// Mitsubishi GX Works2 project: GBOV-76_20100001_210617 H   PLC: Q06UDV
// 21/3/19(五)_進料手臂/開爪修正_

PROGRAM SERVO
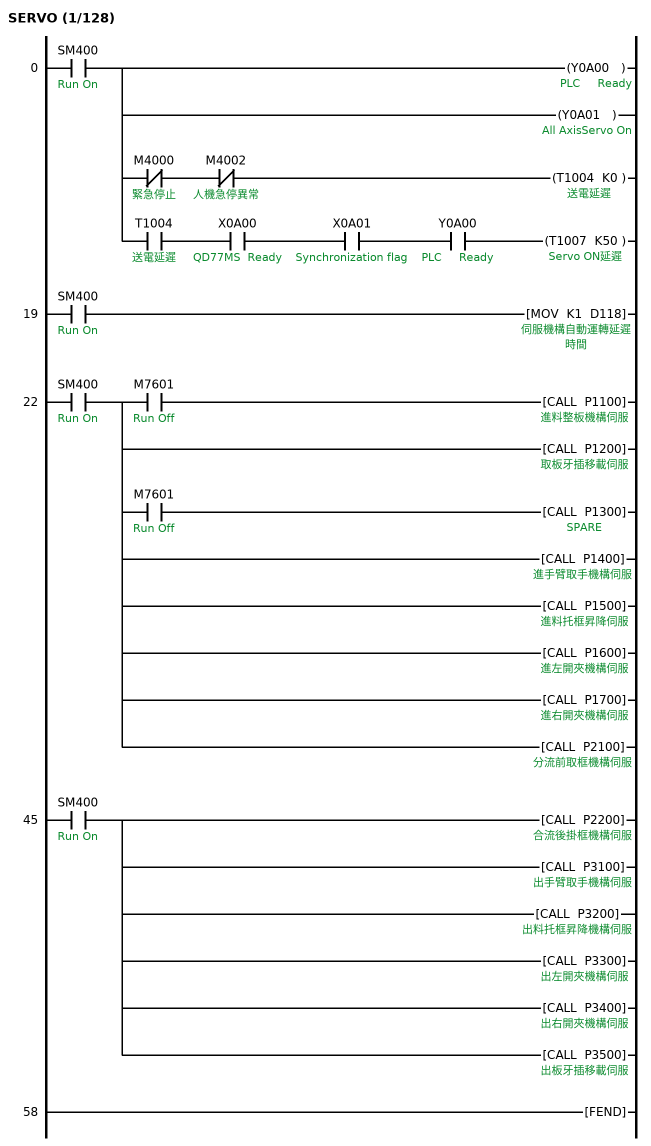
0     LD      SM400  ; Run On
      OUT     Y0A00  ; PLC     Ready
      OUT     Y0A01  ; All AxisServo On
      MPS
      ANI     M4000  ; 緊急停止
      ANI     M4002  ; 人機急停異常
      OUT     T1004 K0  ; 送電延遲
      MPP
      AND     T1004  ; 送電延遲
      AND     X0A00  ; QD77MS  Ready
      AND     X0A01  ; Synchronization flag
      AND     Y0A00  ; PLC     Ready
      OUT     T1007 K50  ; Servo ON延遲
19    LD      SM400  ; Run On
      MOV     K1 D118  ; 伺服機構自動運轉延遲時間
22    LD      SM400  ; Run On
      MPS
      AND     M7601  ; Run Off
      CALL    P1100  ; 進料整板機構伺服
      MPP
      CALL    P1200  ; 取板牙插移載伺服
      MPS
      AND     M7601  ; Run Off
      CALL    P1300  ; SPARE
      MPP
      CALL    P1400  ; 進手臂取手機構伺服
      CALL    P1500  ; 進料托框昇降伺服
      CALL    P1600  ; 進左開夾機構伺服
      CALL    P1700  ; 進右開夾機構伺服
      CALL    P2100  ; 分流前取框機構伺服
45    LD      SM400  ; Run On
      CALL    P2200  ; 合流後掛框機構伺服
      CALL    P3100  ; 出手臂取手機構伺服
      CALL    P3200  ; 出料托框昇降機構伺服
      CALL    P3300  ; 出左開夾機構伺服
      CALL    P3400  ; 出右開夾機構伺服
      CALL    P3500  ; 出板牙插移載伺服
58    FEND
      P1100
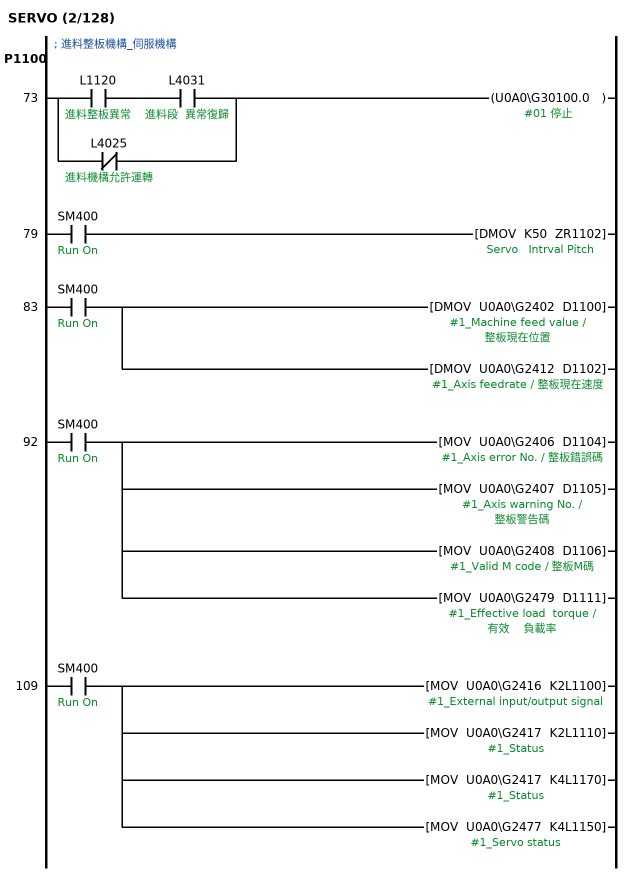
; 進料整板機構_伺服機構
73    LD      L1120  ; 進料整板異常
      AND     L4031  ; 進料段  異常復歸
      ORI     L4025  ; 進料機構允許運轉
      OUT     U0A0\G30100.0  ; #01 停止
79    LD      SM400  ; Run On
      DMOV    K50 ZR1102  ; Servo   Intrval Pitch
83    LD      SM400  ; Run On
      DMOV    U0A0\G2402 D1100  ; #1_Machine feed value / 整板現在位置
      DMOV    U0A0\G2412 D1102  ; #1_Axis feedrate / 整板現在速度
92    LD      SM400  ; Run On
      MOV     U0A0\G2406 D1104  ; #1_Axis error No. / 整板錯誤碼
      MOV     U0A0\G2407 D1105  ; #1_Axis warning No. / 整板警告碼
      MOV     U0A0\G2408 D1106  ; #1_Valid M code / 整板M碼
      MOV     U0A0\G2479 D1111  ; #1_Effective load  torque / 有效    負載率
109   LD      SM400  ; Run On
      MOV     U0A0\G2416 K2L1100  ; #1_External input/output signal / 整板 負極限
      MOV     U0A0\G2417 K2L1110  ; #1_Status / 整板速度控制
      MOV     U0A0\G2417 K4L1170  ; 整板速度控制
      MOV     U0A0\G2477 K4L1150  ; #1_Servo status / READY ON
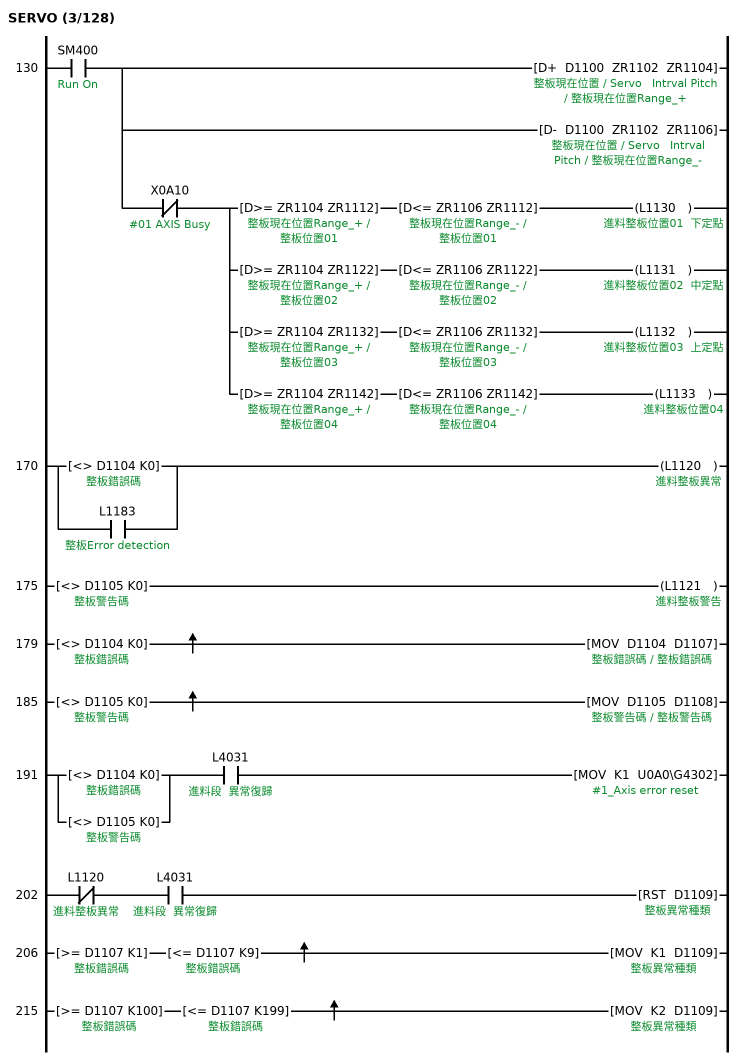
130   LD      SM400  ; Run On
      D+      D1100 ZR1102 ZR1104  ; 整板現在位置Range_+
      D-      D1100 ZR1102 ZR1106  ; 整板現在位置Range_-
      ANI     X0A10  ; #01 AXIS Busy
      MPS
      ANDD>=  ZR1104 ZR1112  ; 整板現在位置Range_+ / 整板位置01
      ANDD<=  ZR1106 ZR1112  ; 整板現在位置Range_- / 整板位置01
      OUT     L1130  ; 進料整板位置01  下定點
      MRD
      ANDD>=  ZR1104 ZR1122  ; 整板現在位置Range_+ / 整板位置02
      ANDD<=  ZR1106 ZR1122  ; 整板現在位置Range_- / 整板位置02
      OUT     L1131  ; 進料整板位置02  中定點
      MRD
      ANDD>=  ZR1104 ZR1132  ; 整板現在位置Range_+ / 整板位置03
      ANDD<=  ZR1106 ZR1132  ; 整板現在位置Range_- / 整板位置03
      OUT     L1132  ; 進料整板位置03  上定點
      MPP
      ANDD>=  ZR1104 ZR1142  ; 整板現在位置Range_+ / 整板位置04
      ANDD<=  ZR1106 ZR1142  ; 整板現在位置Range_- / 整板位置04
      OUT     L1133  ; 進料整板位置04
170   LD<>    D1104 K0  ; 整板錯誤碼
      OR      L1183  ; 整板Error detection
      OUT     L1120  ; 進料整板異常
175   LD<>    D1105 K0  ; 整板警告碼
      OUT     L1121  ; 進料整板警告
179   LD<>    D1104 K0  ; 整板錯誤碼
      MEP
      MOV     D1104 D1107  ; 整板錯誤碼
185   LD<>    D1105 K0  ; 整板警告碼
      MEP
      MOV     D1105 D1108  ; 整板警告碼
191   LD<>    D1104 K0  ; 整板錯誤碼
      OR<>    D1105 K0  ; 整板警告碼
      AND     L4031  ; 進料段  異常復歸
      MOV     K1 U0A0\G4302  ; #1_Axis error reset
202   LDI     L1120  ; 進料整板異常
      AND     L4031  ; 進料段  異常復歸
      RST     D1109  ; 整板異常種類
206   LD>=    D1107 K1  ; 整板錯誤碼
      AND<=   D1107 K9  ; 整板錯誤碼
      MEP
      MOV     K1 D1109
215   LD>=    D1107 K100  ; 整板錯誤碼
      AND<=   D1107 K199  ; 整板錯誤碼
      MEP
      MOV     K2 D1109
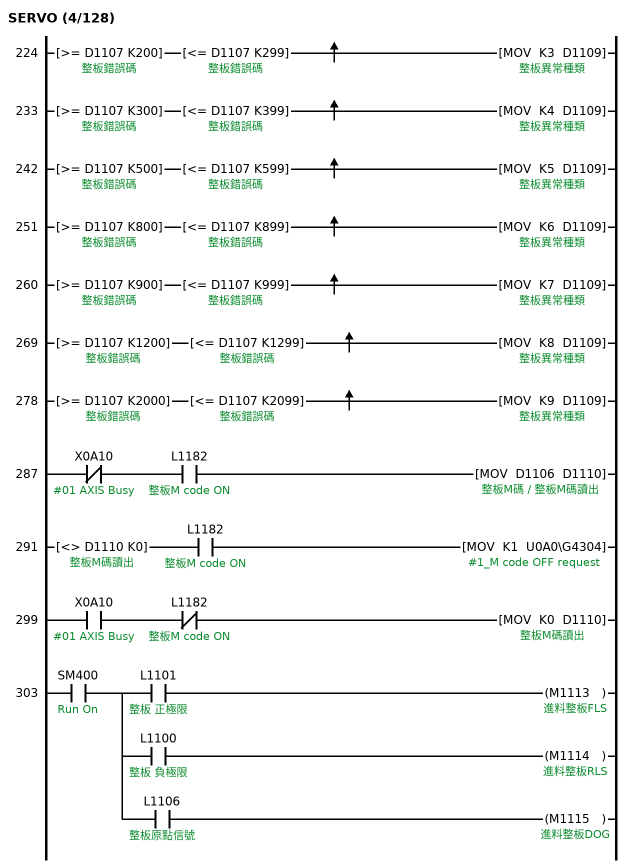
224   LD>=    D1107 K200  ; 整板錯誤碼
      AND<=   D1107 K299  ; 整板錯誤碼
      MEP
      MOV     K3 D1109
233   LD>=    D1107 K300  ; 整板錯誤碼
      AND<=   D1107 K399  ; 整板錯誤碼
      MEP
      MOV     K4 D1109
242   LD>=    D1107 K500  ; 整板錯誤碼
      AND<=   D1107 K599  ; 整板錯誤碼
      MEP
      MOV     K5 D1109
251   LD>=    D1107 K800  ; 整板錯誤碼
      AND<=   D1107 K899  ; 整板錯誤碼
      MEP
      MOV     K6 D1109
260   LD>=    D1107 K900  ; 整板錯誤碼
      AND<=   D1107 K999  ; 整板錯誤碼
      MEP
      MOV     K7 D1109
269   LD>=    D1107 K1200  ; 整板錯誤碼
      AND<=   D1107 K1299  ; 整板錯誤碼
      MEP
      MOV     K8 D1109
278   LD>=    D1107 K2000  ; 整板錯誤碼
      AND<=   D1107 K2099  ; 整板錯誤碼
      MEP
      MOV     K9 D1109
287   LDI     X0A10  ; #01 AXIS Busy
      AND     L1182  ; 整板M code ON
      MOV     D1106 D1110  ; 整板M碼讀出
291   LD<>    D1110 K0  ; 整板M碼讀出
      AND     L1182  ; 整板M code ON
      MOV     K1 U0A0\G4304  ; #1_M code OFF request
299   LD      X0A10  ; #01 AXIS Busy
      ANI     L1182  ; 整板M code ON
      MOV     K0 D1110
303   LD      SM400  ; Run On
      MPS
      AND     L1101  ; 整板 正極限
      OUT     M1113  ; 進料整板FLS
      MRD
      AND     L1100  ; 整板 負極限
      OUT     M1114  ; 進料整板RLS
      MPP
      AND     L1106  ; 整板原點信號
      OUT     M1115  ; 進料整板DOG
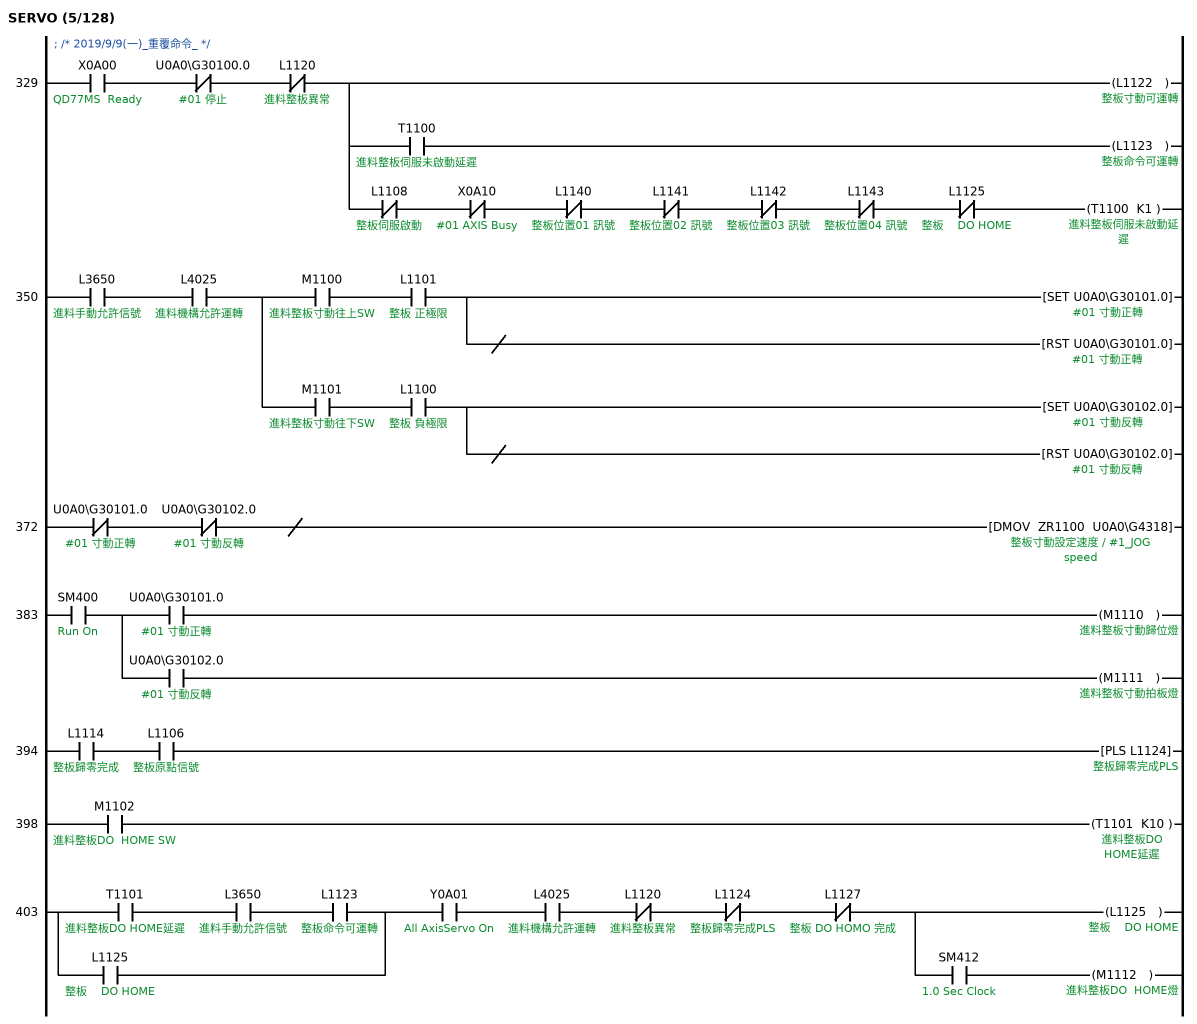
; /* 2019/9/9(一)_重覆命令_ */
329   LD      X0A00  ; QD77MS  Ready
      ANI     U0A0\G30100.0  ; #01 停止
      ANI     L1120  ; 進料整板異常
      OUT     L1122  ; 整板寸動可運轉
      MPS
      AND     T1100  ; 進料整板伺服未啟動延遲
      OUT     L1123  ; 整板命令可運轉
      MPP
      ANI     L1108  ; 整板伺服啟動
      ANI     X0A10  ; #01 AXIS Busy
      ANI     L1140  ; 整板位置01 訊號
      ANI     L1141  ; 整板位置02 訊號
      ANI     L1142  ; 整板位置03 訊號
      ANI     L1143  ; 整板位置04 訊號
      ANI     L1125  ; 整板    DO HOME
      OUT     T1100 K1  ; 進料整板伺服未啟動延遲
350   LD      L3650  ; 進料手動允許信號
      AND     L4025  ; 進料機構允許運轉
      MPS
      AND     M1100  ; 進料整板寸動往上SW
      AND     L1101  ; 整板 正極限
      SET     U0A0\G30101.0  ; #01 寸動正轉
      INV
      RST     U0A0\G30101.0  ; #01 寸動正轉
      MPP
      AND     M1101  ; 進料整板寸動往下SW
      AND     L1100  ; 整板 負極限
      SET     U0A0\G30102.0  ; #01 寸動反轉
      INV
      RST     U0A0\G30102.0  ; #01 寸動反轉
372   LDI     U0A0\G30101.0  ; #01 寸動正轉
      ANI     U0A0\G30102.0  ; #01 寸動反轉
      INV
      DMOV    ZR1100 U0A0\G4318  ; 整板寸動設定速度 / #1_JOG     speed
383   LD      SM400  ; Run On
      MPS
      AND     U0A0\G30101.0  ; #01 寸動正轉
      OUT     M1110  ; 進料整板寸動歸位燈
      MPP
      AND     U0A0\G30102.0  ; #01 寸動反轉
      OUT     M1111  ; 進料整板寸動拍板燈
394   LD      L1114  ; 整板歸零完成
      AND     L1106  ; 整板原點信號
      PLS     L1124  ; 整板歸零完成PLS
398   LD      M1102  ; 進料整板DO  HOME SW
      OUT     T1101 K10  ; 進料整板DO HOME延遲
403   LD      T1101  ; 進料整板DO HOME延遲
      AND     L3650  ; 進料手動允許信號
      AND     L1123  ; 整板命令可運轉
      OR      L1125  ; 整板    DO HOME
      AND     Y0A01  ; All AxisServo On
      AND     L4025  ; 進料機構允許運轉
      ANI     L1120  ; 進料整板異常
      ANI     L1124  ; 整板歸零完成PLS
      ANI     L1127  ; 整板 DO HOMO 完成
      OUT     L1125  ; 整板    DO HOME
      AND     SM412  ; 1.0 Sec Clock
      OUT     M1112  ; 進料整板DO  HOME燈
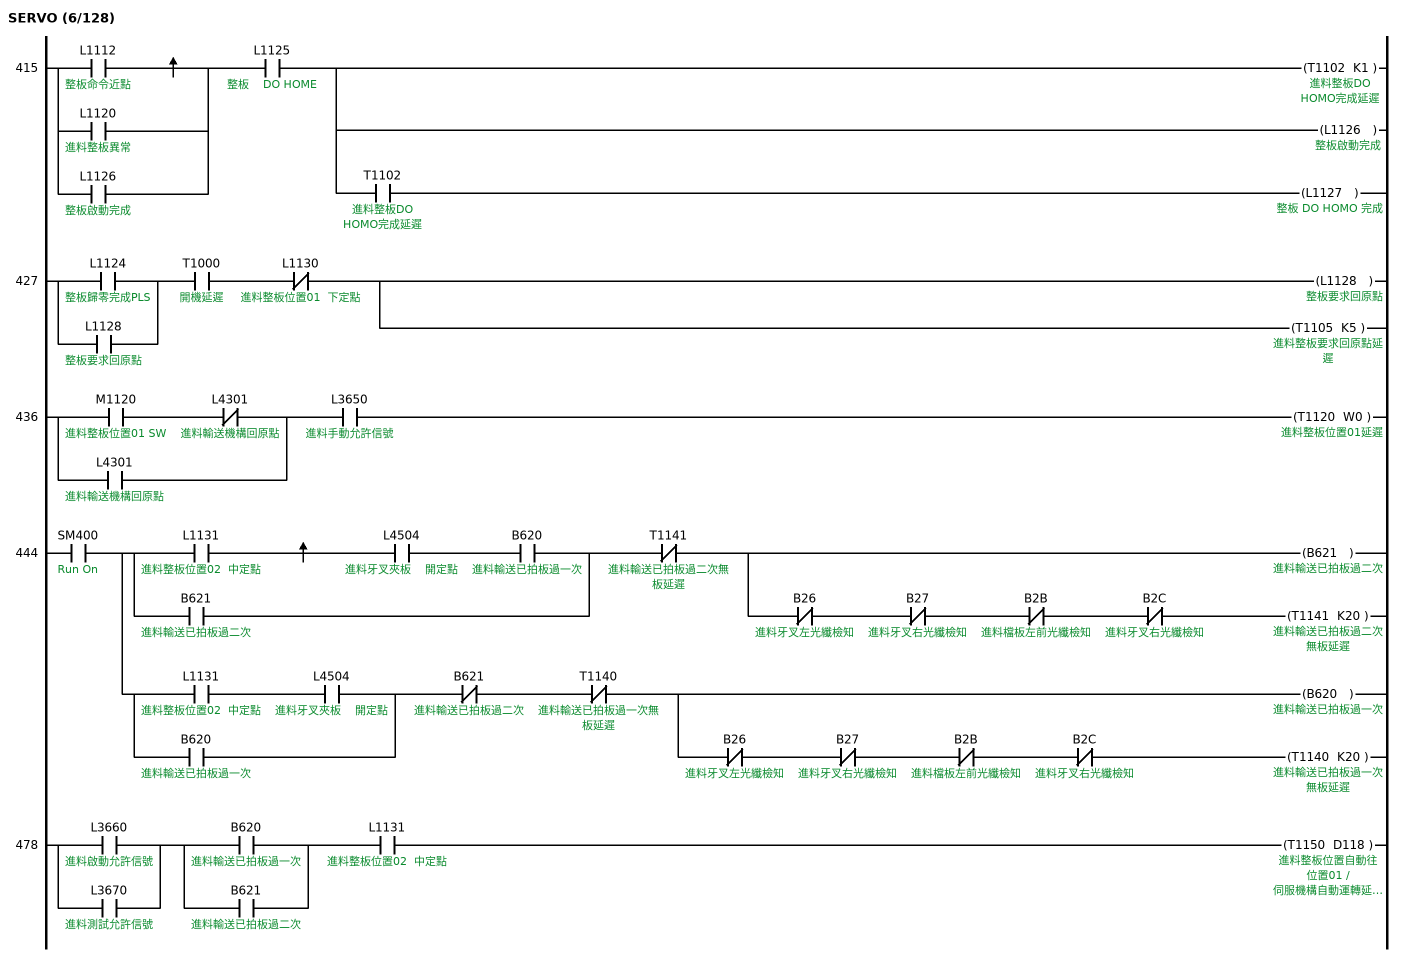
415   LD      L1112  ; 整板命令近點
      MEP
      OR      L1120  ; 進料整板異常
      OR      L1126  ; 整板啟動完成
      AND     L1125  ; 整板    DO HOME
      OUT     T1102 K1  ; 進料整板DO HOMO完成延遲
      OUT     L1126  ; 整板啟動完成
      AND     T1102  ; 進料整板DO HOMO完成延遲
      OUT     L1127  ; 整板 DO HOMO 完成
427   LD      L1124  ; 整板歸零完成PLS
      OR      L1128  ; 整板要求回原點
      AND     T1000  ; 開機延遲
      ANI     L1130  ; 進料整板位置01  下定點
      OUT     L1128  ; 整板要求回原點
      OUT     T1105 K5  ; 進料整板要求回原點延遲
436   LD      M1120  ; 進料整板位置01 SW
      ANI     L4301  ; 進料輸送機構回原點
      OR      L4301  ; 進料輸送機構回原點
      AND     L3650  ; 進料手動允許信號
      OUT     T1120 W0  ; 進料整板位置01延遲
444   LD      SM400  ; Run On
      MPS
      LD      L1131  ; 進料整板位置02  中定點
      MEP
      AND     L4504  ; 進料牙叉夾板    開定點
      AND     B620  ; 進料輸送已拍板過一次
      OR      B621  ; 進料輸送已拍板過二次
      ANB
      ANI     T1141  ; 進料輸送已拍板過二次無板延遲
      OUT     B621  ; 進料輸送已拍板過二次
      ANI     B26  ; 進料牙叉左光纖檢知
      ANI     B27  ; 進料牙叉右光纖檢知
      ANI     B2B  ; 進料檔板左前光纖檢知
      ANI     B2C  ; 進料牙叉右光纖檢知
      OUT     T1141 K20  ; 進料輸送已拍板過二次無板延遲
      MPP
      LD      L1131  ; 進料整板位置02  中定點
      AND     L4504  ; 進料牙叉夾板    開定點
      OR      B620  ; 進料輸送已拍板過一次
      ANB
      ANI     B621  ; 進料輸送已拍板過二次
      ANI     T1140  ; 進料輸送已拍板過一次無板延遲
      OUT     B620  ; 進料輸送已拍板過一次
      ANI     B26  ; 進料牙叉左光纖檢知
      ANI     B27  ; 進料牙叉右光纖檢知
      ANI     B2B  ; 進料檔板左前光纖檢知
      ANI     B2C  ; 進料牙叉右光纖檢知
      OUT     T1140 K20  ; 進料輸送已拍板過一次無板延遲
478   LD      L3660  ; 進料啟動允許信號
      OR      L3670  ; 進料測試允許信號
      LD      B620  ; 進料輸送已拍板過一次
      OR      B621  ; 進料輸送已拍板過二次
      ANB
      AND     L1131  ; 進料整板位置02  中定點
      OUT     T1150 D118  ; 進料整板位置自動往  位置01 / 伺服機構自動運轉延遲時間
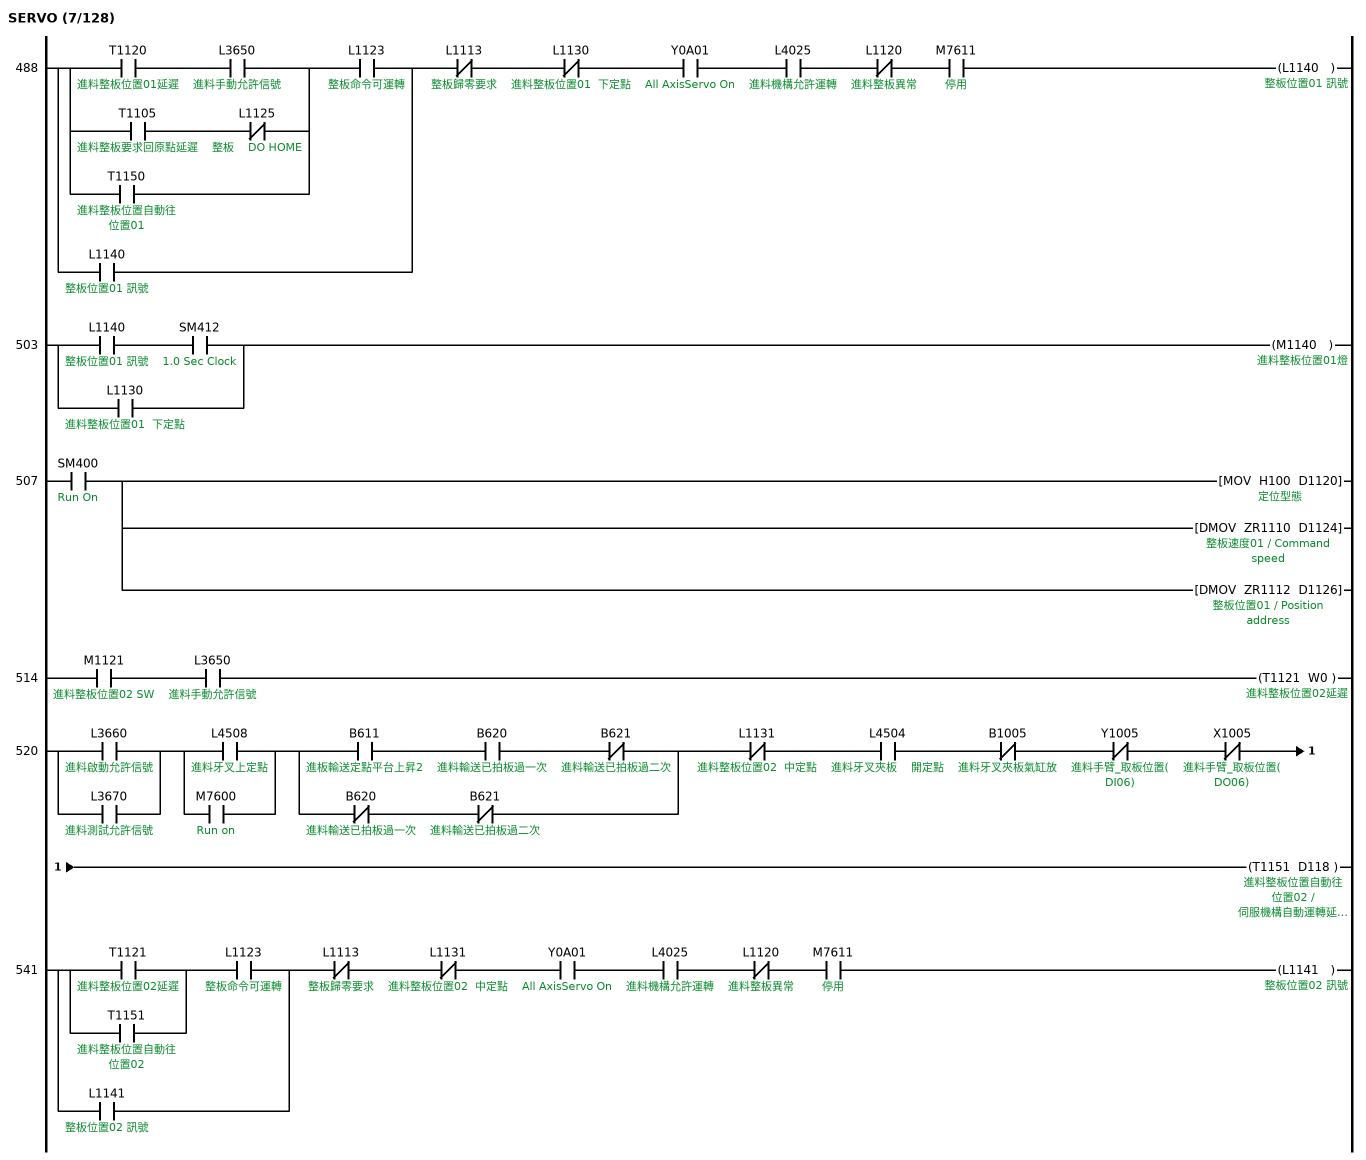
488   LD      T1120  ; 進料整板位置01延遲
      AND     L3650  ; 進料手動允許信號
      LD      T1105  ; 進料整板要求回原點延遲
      ANI     L1125  ; 整板    DO HOME
      ORB
      OR      T1150  ; 進料整板位置自動往  位置01
      AND     L1123  ; 整板命令可運轉
      OR      L1140  ; 整板位置01 訊號
      ANI     L1113  ; 整板歸零要求
      ANI     L1130  ; 進料整板位置01  下定點
      AND     Y0A01  ; All AxisServo On
      AND     L4025  ; 進料機構允許運轉
      ANI     L1120  ; 進料整板異常
      AND     M7611  ; 停用
      OUT     L1140  ; 整板位置01 訊號
503   LD      L1140  ; 整板位置01 訊號
      AND     SM412  ; 1.0 Sec Clock
      OR      L1130  ; 進料整板位置01  下定點
      OUT     M1140  ; 進料整板位置01燈
507   LD      SM400  ; Run On
      MOV     H100 D1120  ; 定位型態
      DMOV    ZR1110 D1124  ; 整板速度01 / Command  speed
      DMOV    ZR1112 D1126  ; Position address
514   LD      M1121  ; 進料整板位置02 SW
      AND     L3650  ; 進料手動允許信號
      OUT     T1121 W0  ; 進料整板位置02延遲
520   LD      L3660  ; 進料啟動允許信號
      OR      L3670  ; 進料測試允許信號
      LD      L4508  ; 進料牙叉上定點
      OR      M7600  ; Run on
      ANB
      LD      B611  ; 進板輸送定點平台上昇2
      AND     B620  ; 進料輸送已拍板過一次
      ANI     B621  ; 進料輸送已拍板過二次
      LDI     B620  ; 進料輸送已拍板過一次
      ANI     B621  ; 進料輸送已拍板過二次
      ORB
      ANB
      ANI     L1131  ; 進料整板位置02  中定點
      AND     L4504  ; 進料牙叉夾板    開定點
      ANI     B1005  ; 進料牙叉夾板氣缸放
      ANI     Y1005  ; 進料手臂_取板位置(DI06)
      ANI     X1005  ; 進料手臂_取板位置(DO06)
      OUT     T1151 D118  ; 進料整板位置自動往  位置02 / 伺服機構自動運轉延遲時間
541   LD      T1121  ; 進料整板位置02延遲
      OR      T1151  ; 進料整板位置自動往  位置02
      AND     L1123  ; 整板命令可運轉
      OR      L1141  ; 整板位置02 訊號
      ANI     L1113  ; 整板歸零要求
      ANI     L1131  ; 進料整板位置02  中定點
      AND     Y0A01  ; All AxisServo On
      AND     L4025  ; 進料機構允許運轉
      ANI     L1120  ; 進料整板異常
      AND     M7611  ; 停用
      OUT     L1141  ; 整板位置02 訊號
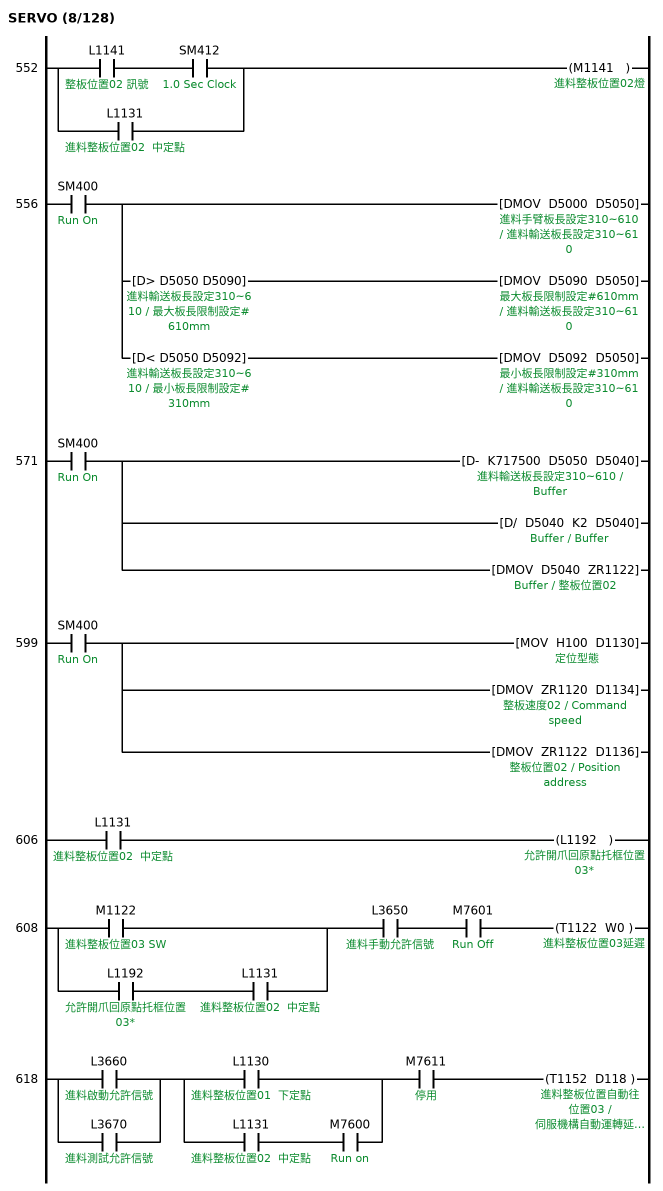
552   LD      L1141  ; 整板位置02 訊號
      AND     SM412  ; 1.0 Sec Clock
      OR      L1131  ; 進料整板位置02  中定點
      OUT     M1141  ; 進料整板位置02燈
556   LD      SM400  ; Run On
      DMOV    D5000 D5050  ; 進料手臂板長設定310~610 / 進料輸送板長設定310~610
      MPS
      ANDD>   D5050 D5090  ; 進料輸送板長設定310~610 / 最大板長限制設定#610mm
      DMOV    D5090 D5050
      MPP
      ANDD<   D5050 D5092  ; 進料輸送板長設定310~610 / 最小板長限制設定#310mm
      DMOV    D5092 D5050
571   LD      SM400  ; Run On
      D-      K717500 D5050 D5040  ; Buffer
        [note] /* 輸送拍板原點尺寸_717.5mm */
      D/      D5040 K2 D5040
      DMOV    D5040 ZR1122
599   LD      SM400  ; Run On
      MOV     H100 D1130  ; 定位型態
      DMOV    ZR1120 D1134  ; 整板速度02 / Command  speed
      DMOV    ZR1122 D1136  ; Position address
606   LD      L1131  ; 進料整板位置02  中定點
      OUT     L1192  ; 允許開爪回原點托框位置03*
608   LD      M1122  ; 進料整板位置03 SW
      LD      L1192  ; 允許開爪回原點托框位置03*
      AND     L1131  ; 進料整板位置02  中定點
      ORB
      AND     L3650  ; 進料手動允許信號
      AND     M7601  ; Run Off
      OUT     T1122 W0  ; 進料整板位置03延遲
618   LD      L3660  ; 進料啟動允許信號
      OR      L3670  ; 進料測試允許信號
      LD      L1130  ; 進料整板位置01  下定點
      LD      L1131  ; 進料整板位置02  中定點
      AND     M7600  ; Run on
      ORB
      ANB
      AND     M7611  ; 停用
      OUT     T1152 D118  ; 進料整板位置自動往  位置03 / 伺服機構自動運轉延遲時間
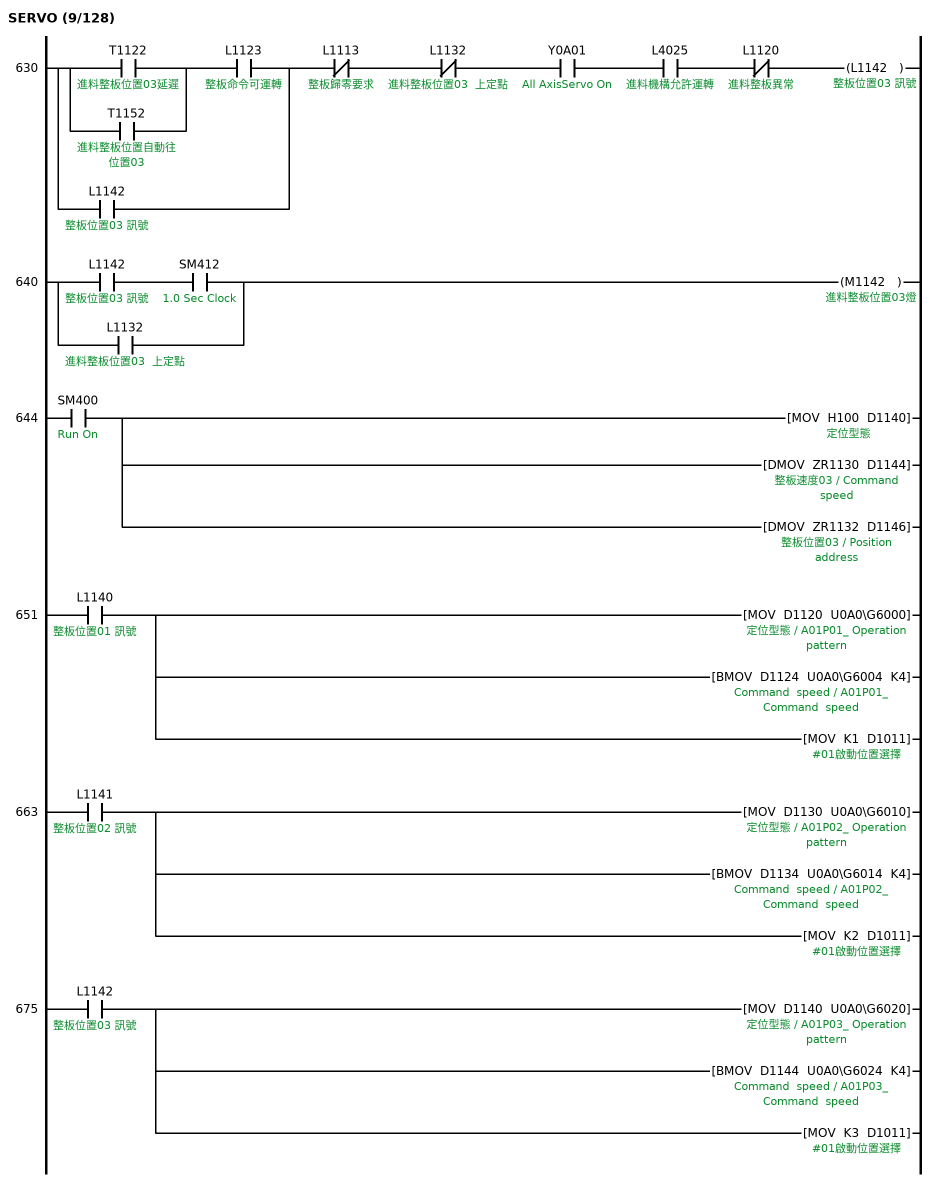
630   LD      T1122  ; 進料整板位置03延遲
      OR      T1152  ; 進料整板位置自動往  位置03
      AND     L1123  ; 整板命令可運轉
      OR      L1142  ; 整板位置03 訊號
      ANI     L1113  ; 整板歸零要求
      ANI     L1132  ; 進料整板位置03  上定點
      AND     Y0A01  ; All AxisServo On
      AND     L4025  ; 進料機構允許運轉
      ANI     L1120  ; 進料整板異常
      OUT     L1142  ; 整板位置03 訊號
640   LD      L1142  ; 整板位置03 訊號
      AND     SM412  ; 1.0 Sec Clock
      OR      L1132  ; 進料整板位置03  上定點
      OUT     M1142  ; 進料整板位置03燈
644   LD      SM400  ; Run On
      MOV     H100 D1140  ; 定位型態
      DMOV    ZR1130 D1144  ; 整板速度03 / Command  speed
      DMOV    ZR1132 D1146  ; Position address
651   LD      L1140  ; 整板位置01 訊號
      MOV     D1120 U0A0\G6000  ; A01P01_ Operation pattern
      BMOV    D1124 U0A0\G6004 K4  ; A01P01_ Command  speed
      MOV     K1 D1011  ; #01啟動位置選擇
663   LD      L1141  ; 整板位置02 訊號
      MOV     D1130 U0A0\G6010  ; A01P02_ Operation pattern
      BMOV    D1134 U0A0\G6014 K4  ; A01P02_ Command  speed
      MOV     K2 D1011
675   LD      L1142  ; 整板位置03 訊號
      MOV     D1140 U0A0\G6020  ; A01P03_ Operation pattern
      BMOV    D1144 U0A0\G6024 K4  ; A01P03_ Command  speed
      MOV     K3 D1011
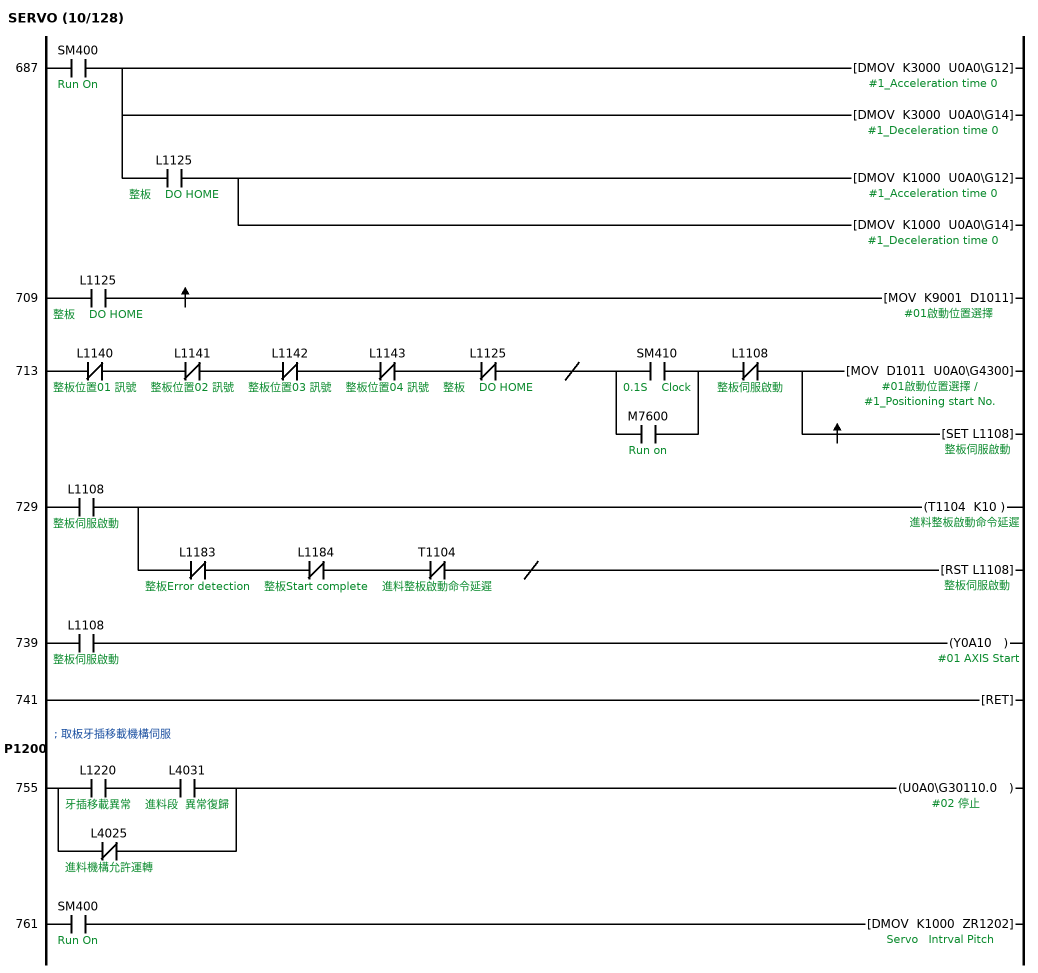
687   LD      SM400  ; Run On
      DMOV    K3000 U0A0\G12  ; #1_Acceleration time 0
      DMOV    K3000 U0A0\G14  ; #1_Deceleration time 0
      AND     L1125  ; 整板    DO HOME
      DMOV    K1000 U0A0\G12
      DMOV    K1000 U0A0\G14
709   LD      L1125  ; 整板    DO HOME
      MEP
      MOV     K9001 D1011
713   LDI     L1140  ; 整板位置01 訊號
      ANI     L1141  ; 整板位置02 訊號
      ANI     L1142  ; 整板位置03 訊號
      ANI     L1143  ; 整板位置04 訊號
      ANI     L1125  ; 整板    DO HOME
      INV
      LD      SM410  ; 0.1S    Clock
      OR      M7600  ; Run on
      ANB
      ANI     L1108  ; 整板伺服啟動
      MOV     D1011 U0A0\G4300  ; #1_Positioning start No.
      MEP
      SET     L1108  ; 整板伺服啟動
729   LD      L1108  ; 整板伺服啟動
      OUT     T1104 K10  ; 進料整板啟動命令延遲
      ANI     L1183  ; 整板Error detection
      ANI     L1184  ; 整板Start complete
      ANI     T1104  ; 進料整板啟動命令延遲
      INV
      RST     L1108  ; 整板伺服啟動
739   LD      L1108  ; 整板伺服啟動
      OUT     Y0A10  ; #01 AXIS Start
741   RET
      P1200
; 取板牙插移載機構伺服
755   LD      L1220  ; 牙插移載異常
      AND     L4031  ; 進料段  異常復歸
      ORI     L4025  ; 進料機構允許運轉
      OUT     U0A0\G30110.0  ; #02 停止
761   LD      SM400  ; Run On
      DMOV    K1000 ZR1202  ; Servo   Intrval Pitch
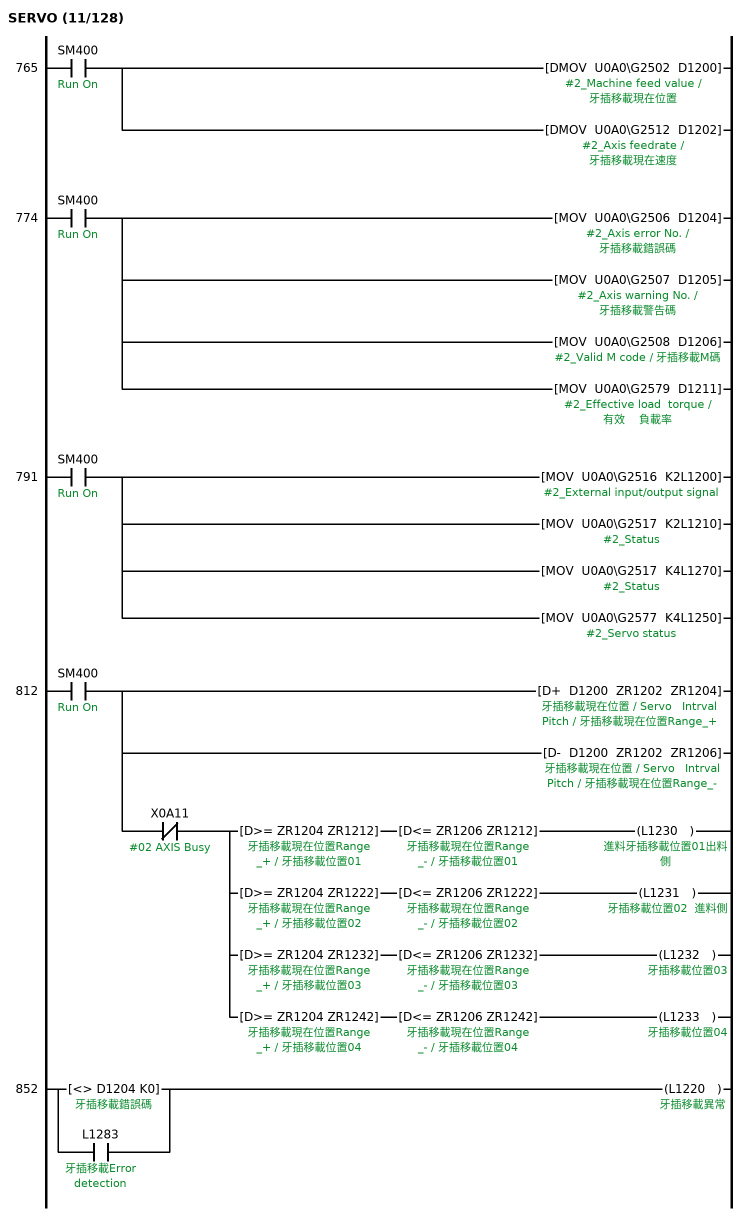
765   LD      SM400  ; Run On
      DMOV    U0A0\G2502 D1200  ; #2_Machine feed value / 牙插移載現在位置
      DMOV    U0A0\G2512 D1202  ; #2_Axis feedrate / 牙插移載現在速度
774   LD      SM400  ; Run On
      MOV     U0A0\G2506 D1204  ; #2_Axis error No. / 牙插移載錯誤碼
      MOV     U0A0\G2507 D1205  ; #2_Axis warning No. / 牙插移載警告碼
      MOV     U0A0\G2508 D1206  ; #2_Valid M code / 牙插移載M碼
      MOV     U0A0\G2579 D1211  ; #2_Effective load  torque / 有效    負載率
791   LD      SM400  ; Run On
      MOV     U0A0\G2516 K2L1200  ; #2_External input/output signal / 牙插移載    負極限
      MOV     U0A0\G2517 K2L1210  ; #2_Status / 牙插移載速度控制
      MOV     U0A0\G2517 K4L1270  ; 牙插移載速度控制
      MOV     U0A0\G2577 K4L1250  ; #2_Servo status / READY ON
812   LD      SM400  ; Run On
      D+      D1200 ZR1202 ZR1204  ; 牙插移載現在位置Range_+
      D-      D1200 ZR1202 ZR1206  ; 牙插移載現在位置Range_-
      ANI     X0A11  ; #02 AXIS Busy
      MPS
      ANDD>=  ZR1204 ZR1212  ; 牙插移載現在位置Range_+ / 牙插移載位置01
      ANDD<=  ZR1206 ZR1212  ; 牙插移載現在位置Range_- / 牙插移載位置01
      OUT     L1230  ; 進料牙插移載位置01出料側
      MRD
      ANDD>=  ZR1204 ZR1222  ; 牙插移載現在位置Range_+ / 牙插移載位置02
      ANDD<=  ZR1206 ZR1222  ; 牙插移載現在位置Range_- / 牙插移載位置02
      OUT     L1231  ; 牙插移載位置02  進料側
      MRD
      ANDD>=  ZR1204 ZR1232  ; 牙插移載現在位置Range_+ / 牙插移載位置03
      ANDD<=  ZR1206 ZR1232  ; 牙插移載現在位置Range_- / 牙插移載位置03
      OUT     L1232  ; 牙插移載位置03
      MPP
      ANDD>=  ZR1204 ZR1242  ; 牙插移載現在位置Range_+ / 牙插移載位置04
      ANDD<=  ZR1206 ZR1242  ; 牙插移載現在位置Range_- / 牙插移載位置04
      OUT     L1233  ; 牙插移載位置04
852   LD<>    D1204 K0  ; 牙插移載錯誤碼
      OR      L1283  ; 牙插移載Error detection
      OUT     L1220  ; 牙插移載異常
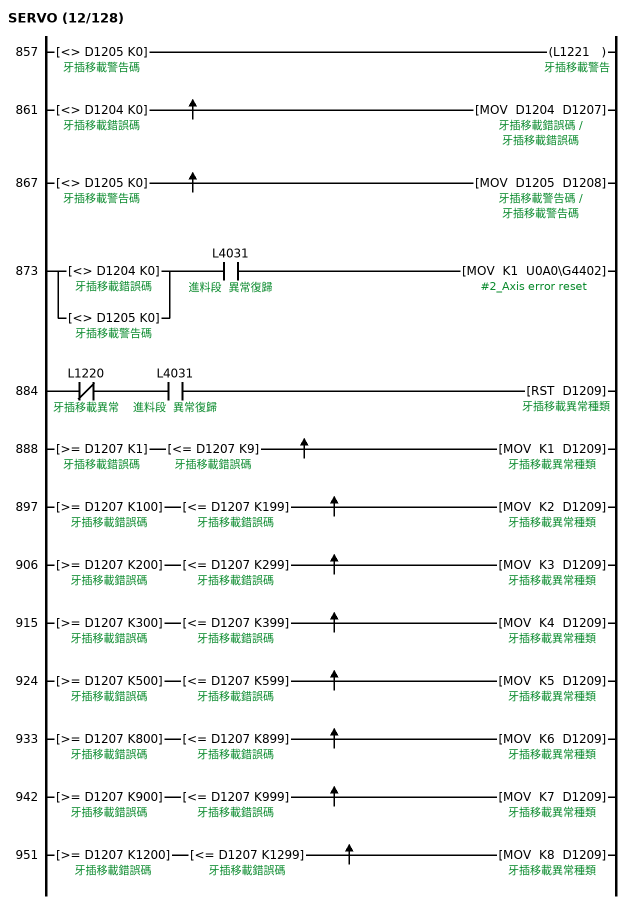
857   LD<>    D1205 K0  ; 牙插移載警告碼
      OUT     L1221  ; 牙插移載警告
861   LD<>    D1204 K0  ; 牙插移載錯誤碼
      MEP
      MOV     D1204 D1207  ; 牙插移載錯誤碼
867   LD<>    D1205 K0  ; 牙插移載警告碼
      MEP
      MOV     D1205 D1208  ; 牙插移載警告碼
873   LD<>    D1204 K0  ; 牙插移載錯誤碼
      OR<>    D1205 K0  ; 牙插移載警告碼
      AND     L4031  ; 進料段  異常復歸
      MOV     K1 U0A0\G4402  ; #2_Axis error reset
884   LDI     L1220  ; 牙插移載異常
      AND     L4031  ; 進料段  異常復歸
      RST     D1209  ; 牙插移載異常種類
888   LD>=    D1207 K1  ; 牙插移載錯誤碼
      AND<=   D1207 K9  ; 牙插移載錯誤碼
      MEP
      MOV     K1 D1209
897   LD>=    D1207 K100  ; 牙插移載錯誤碼
      AND<=   D1207 K199  ; 牙插移載錯誤碼
      MEP
      MOV     K2 D1209
906   LD>=    D1207 K200  ; 牙插移載錯誤碼
      AND<=   D1207 K299  ; 牙插移載錯誤碼
      MEP
      MOV     K3 D1209
915   LD>=    D1207 K300  ; 牙插移載錯誤碼
      AND<=   D1207 K399  ; 牙插移載錯誤碼
      MEP
      MOV     K4 D1209
924   LD>=    D1207 K500  ; 牙插移載錯誤碼
      AND<=   D1207 K599  ; 牙插移載錯誤碼
      MEP
      MOV     K5 D1209
933   LD>=    D1207 K800  ; 牙插移載錯誤碼
      AND<=   D1207 K899  ; 牙插移載錯誤碼
      MEP
      MOV     K6 D1209
942   LD>=    D1207 K900  ; 牙插移載錯誤碼
      AND<=   D1207 K999  ; 牙插移載錯誤碼
      MEP
      MOV     K7 D1209
951   LD>=    D1207 K1200  ; 牙插移載錯誤碼
      AND<=   D1207 K1299  ; 牙插移載錯誤碼
      MEP
      MOV     K8 D1209
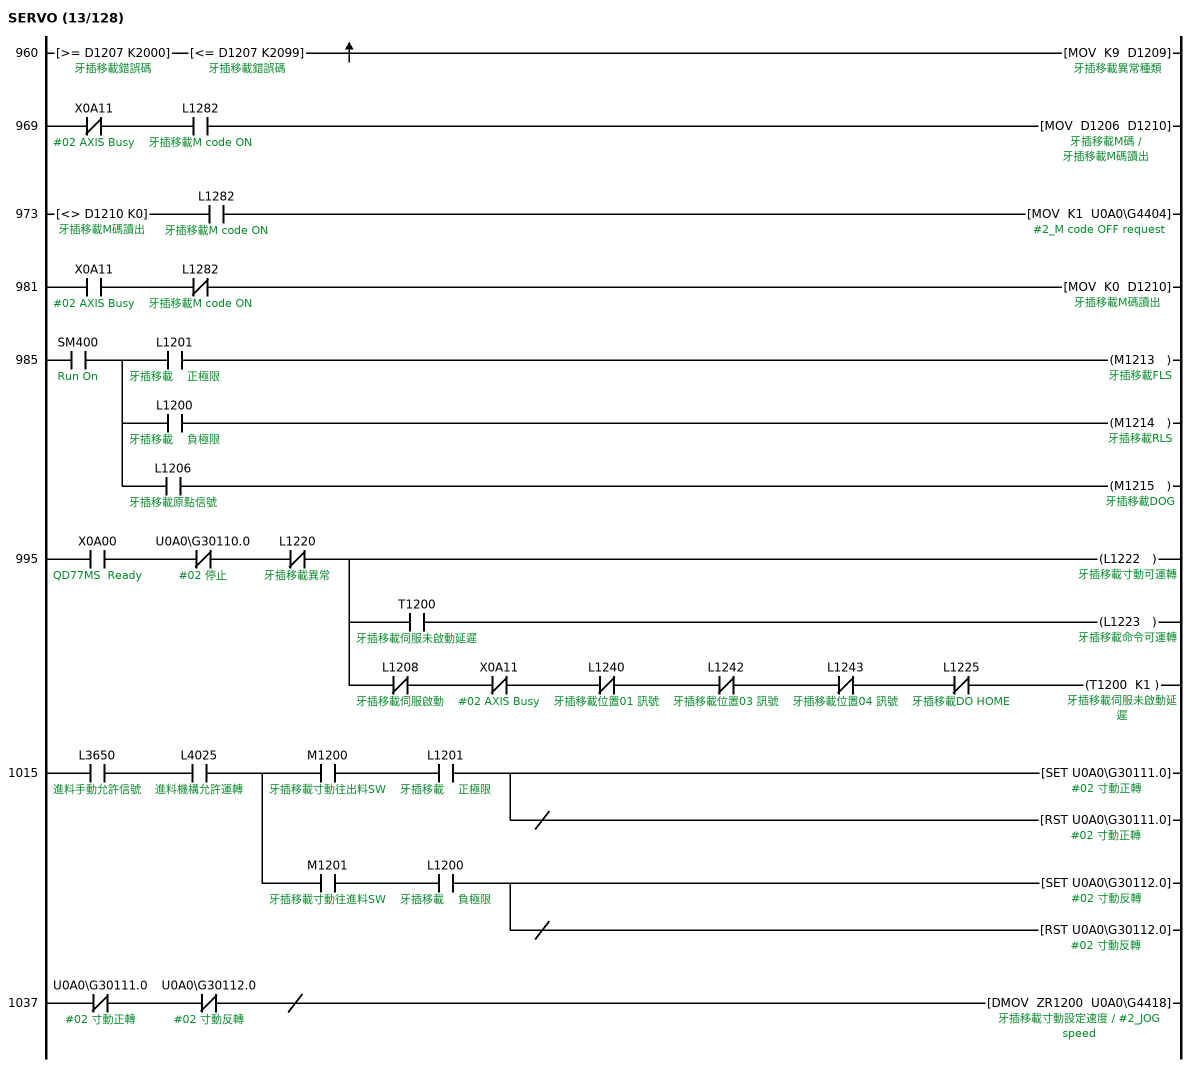
960   LD>=    D1207 K2000  ; 牙插移載錯誤碼
      AND<=   D1207 K2099  ; 牙插移載錯誤碼
      MEP
      MOV     K9 D1209
969   LDI     X0A11  ; #02 AXIS Busy
      AND     L1282  ; 牙插移載M code ON
      MOV     D1206 D1210  ; 牙插移載M碼讀出
973   LD<>    D1210 K0  ; 牙插移載M碼讀出
      AND     L1282  ; 牙插移載M code ON
      MOV     K1 U0A0\G4404  ; #2_M code OFF request
981   LD      X0A11  ; #02 AXIS Busy
      ANI     L1282  ; 牙插移載M code ON
      MOV     K0 D1210
985   LD      SM400  ; Run On
      MPS
      AND     L1201  ; 牙插移載    正極限
      OUT     M1213  ; 牙插移載FLS
      MRD
      AND     L1200  ; 牙插移載    負極限
      OUT     M1214  ; 牙插移載RLS
      MPP
      AND     L1206  ; 牙插移載原點信號
      OUT     M1215  ; 牙插移載DOG
995   LD      X0A00  ; QD77MS  Ready
      ANI     U0A0\G30110.0  ; #02 停止
      ANI     L1220  ; 牙插移載異常
      OUT     L1222  ; 牙插移載寸動可運轉
      MPS
      AND     T1200  ; 牙插移載伺服未啟動延遲
      OUT     L1223  ; 牙插移載命令可運轉
      MPP
      ANI     L1208  ; 牙插移載伺服啟動
      ANI     X0A11  ; #02 AXIS Busy
      ANI     L1240  ; 牙插移載位置01 訊號
      ANI     L1242  ; 牙插移載位置03 訊號
      ANI     L1243  ; 牙插移載位置04 訊號
      ANI     L1225  ; 牙插移載DO HOME
      OUT     T1200 K1  ; 牙插移載伺服未啟動延遲
1015  LD      L3650  ; 進料手動允許信號
      AND     L4025  ; 進料機構允許運轉
      MPS
      AND     M1200  ; 牙插移載寸動往出料SW
      AND     L1201  ; 牙插移載    正極限
      SET     U0A0\G30111.0  ; #02 寸動正轉
      INV
      RST     U0A0\G30111.0  ; #02 寸動正轉
      MPP
      AND     M1201  ; 牙插移載寸動往進料SW
      AND     L1200  ; 牙插移載    負極限
      SET     U0A0\G30112.0  ; #02 寸動反轉
      INV
      RST     U0A0\G30112.0  ; #02 寸動反轉
1037  LDI     U0A0\G30111.0  ; #02 寸動正轉
      ANI     U0A0\G30112.0  ; #02 寸動反轉
      INV
      DMOV    ZR1200 U0A0\G4418  ; 牙插移載寸動設定速度 / #2_JOG     speed
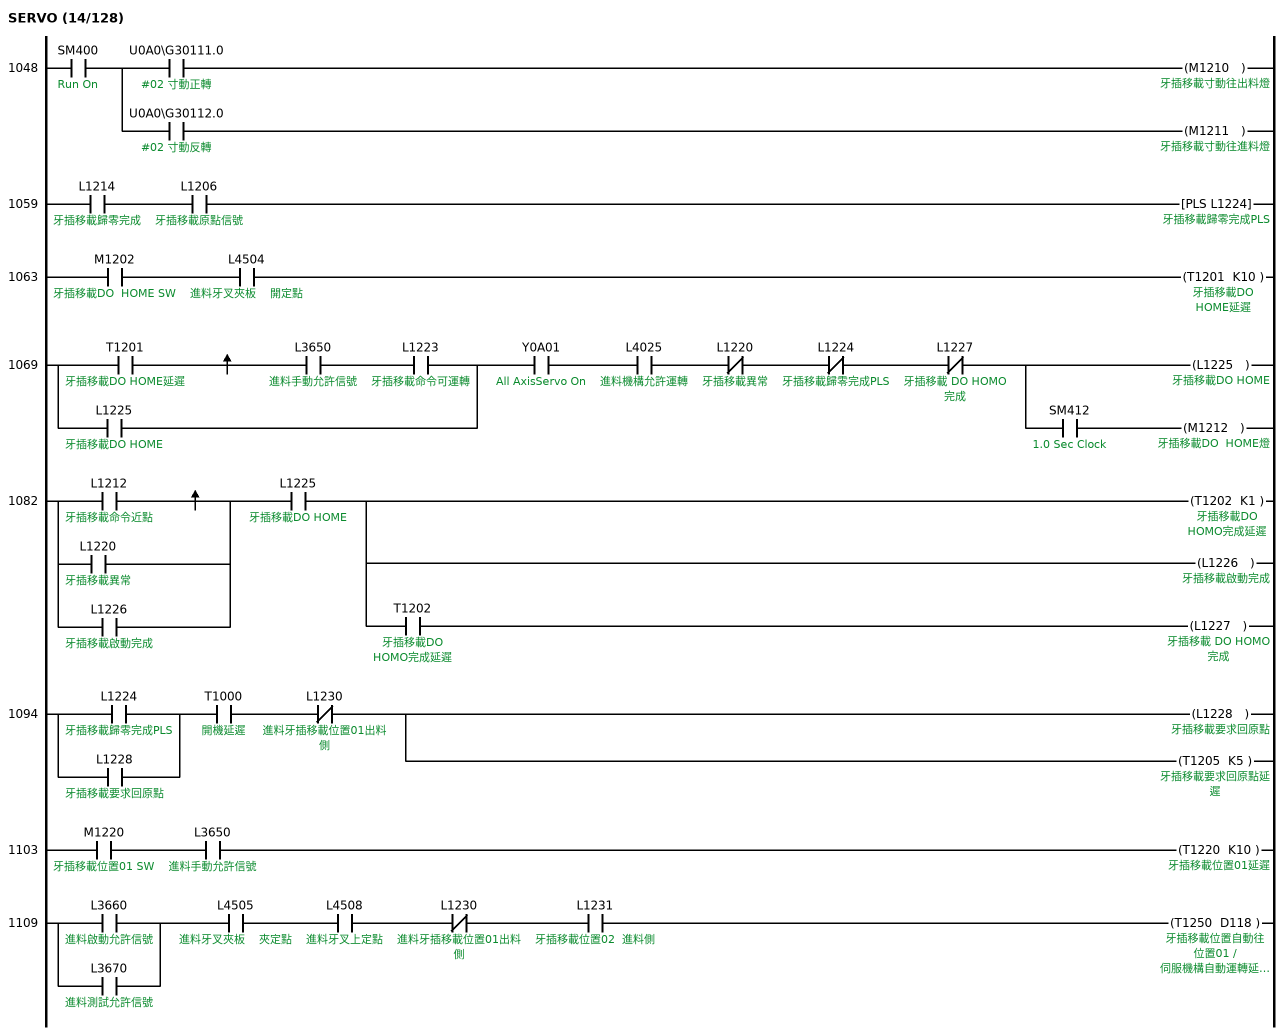
1048  LD      SM400  ; Run On
      MPS
      AND     U0A0\G30111.0  ; #02 寸動正轉
      OUT     M1210  ; 牙插移載寸動往出料燈
      MPP
      AND     U0A0\G30112.0  ; #02 寸動反轉
      OUT     M1211  ; 牙插移載寸動往進料燈
1059  LD      L1214  ; 牙插移載歸零完成
      AND     L1206  ; 牙插移載原點信號
      PLS     L1224  ; 牙插移載歸零完成PLS
1063  LD      M1202  ; 牙插移載DO  HOME SW
      AND     L4504  ; 進料牙叉夾板    開定點
      OUT     T1201 K10  ; 牙插移載DO HOME延遲
1069  LD      T1201  ; 牙插移載DO HOME延遲
      MEP
      AND     L3650  ; 進料手動允許信號
      AND     L1223  ; 牙插移載命令可運轉
      OR      L1225  ; 牙插移載DO HOME
      AND     Y0A01  ; All AxisServo On
      AND     L4025  ; 進料機構允許運轉
      ANI     L1220  ; 牙插移載異常
      ANI     L1224  ; 牙插移載歸零完成PLS
      ANI     L1227  ; 牙插移載 DO HOMO 完成
      OUT     L1225  ; 牙插移載DO HOME
      AND     SM412  ; 1.0 Sec Clock
      OUT     M1212  ; 牙插移載DO  HOME燈
1082  LD      L1212  ; 牙插移載命令近點
      MEP
      OR      L1220  ; 牙插移載異常
      OR      L1226  ; 牙插移載啟動完成
      AND     L1225  ; 牙插移載DO HOME
      OUT     T1202 K1  ; 牙插移載DO HOMO完成延遲
      OUT     L1226  ; 牙插移載啟動完成
      AND     T1202  ; 牙插移載DO HOMO完成延遲
      OUT     L1227  ; 牙插移載 DO HOMO 完成
1094  LD      L1224  ; 牙插移載歸零完成PLS
      OR      L1228  ; 牙插移載要求回原點
      AND     T1000  ; 開機延遲
      ANI     L1230  ; 進料牙插移載位置01出料側
      OUT     L1228  ; 牙插移載要求回原點
      OUT     T1205 K5  ; 牙插移載要求回原點延遲
1103  LD      M1220  ; 牙插移載位置01 SW
      AND     L3650  ; 進料手動允許信號
      OUT     T1220 K10  ; 牙插移載位置01延遲
1109  LD      L3660  ; 進料啟動允許信號
      OR      L3670  ; 進料測試允許信號
      AND     L4505  ; 進料牙叉夾板    夾定點
      AND     L4508  ; 進料牙叉上定點
      ANI     L1230  ; 進料牙插移載位置01出料側
      AND     L1231  ; 牙插移載位置02  進料側
      OUT     T1250 D118  ; 牙插移載位置自動往  位置01 / 伺服機構自動運轉延遲時間
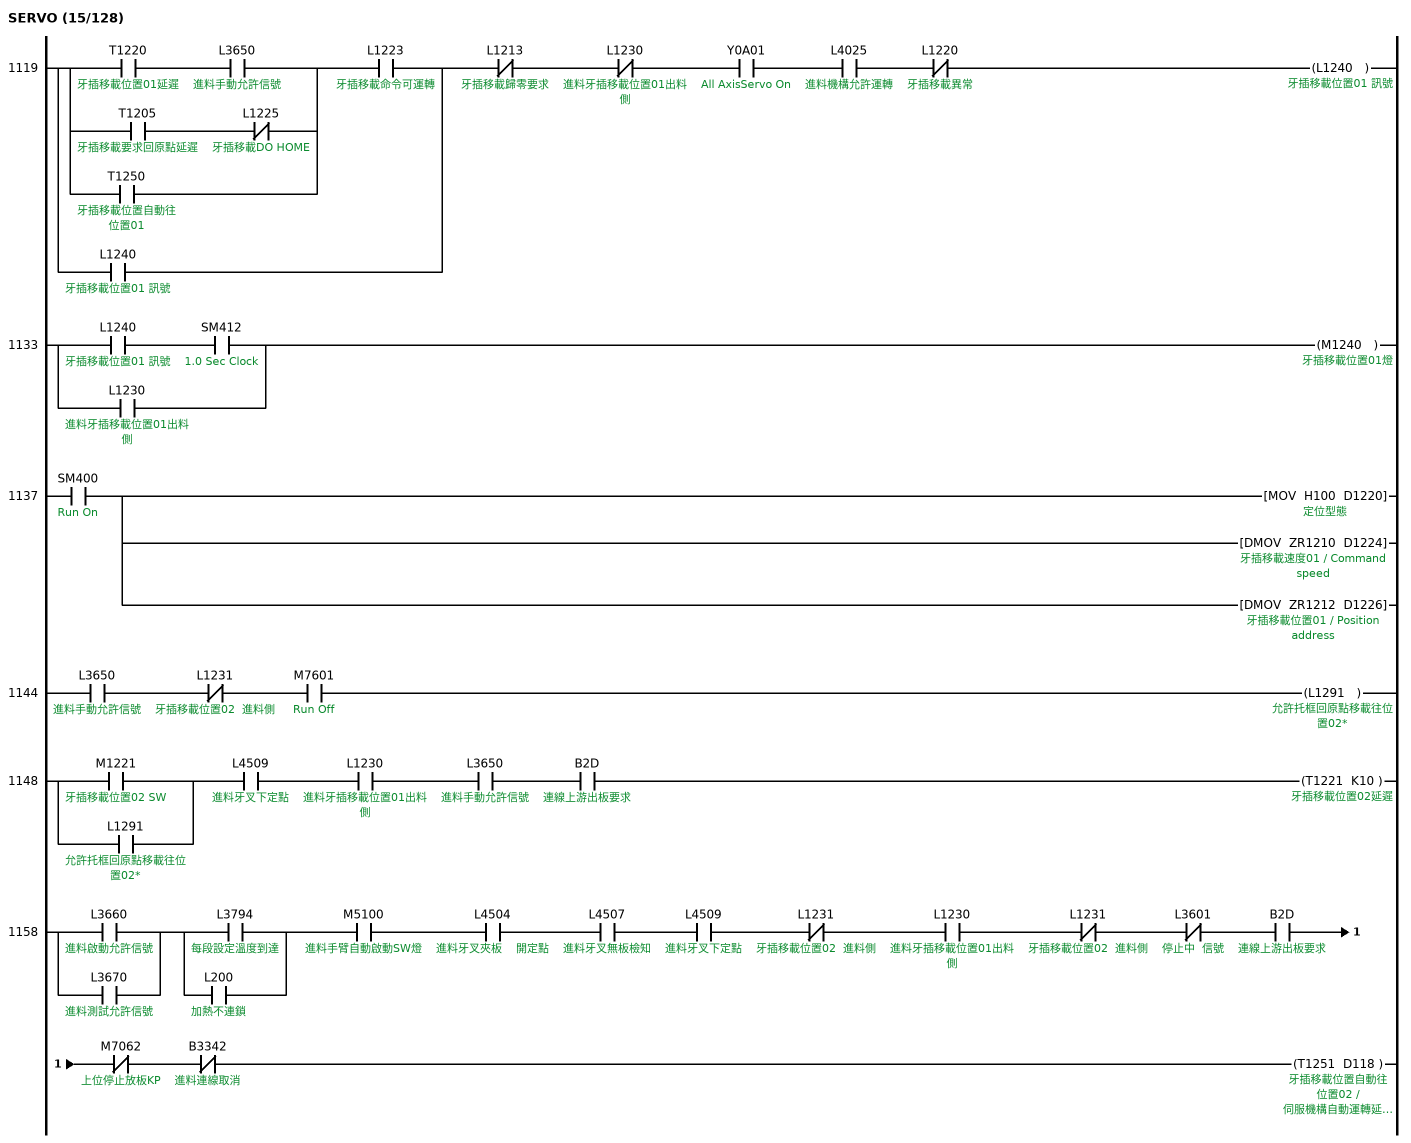
1119  LD      T1220  ; 牙插移載位置01延遲
      AND     L3650  ; 進料手動允許信號
      LD      T1205  ; 牙插移載要求回原點延遲
      ANI     L1225  ; 牙插移載DO HOME
      ORB
      OR      T1250  ; 牙插移載位置自動往  位置01
      AND     L1223  ; 牙插移載命令可運轉
      OR      L1240  ; 牙插移載位置01 訊號
      ANI     L1213  ; 牙插移載歸零要求
      ANI     L1230  ; 進料牙插移載位置01出料側
      AND     Y0A01  ; All AxisServo On
      AND     L4025  ; 進料機構允許運轉
      ANI     L1220  ; 牙插移載異常
      OUT     L1240  ; 牙插移載位置01 訊號
1133  LD      L1240  ; 牙插移載位置01 訊號
      AND     SM412  ; 1.0 Sec Clock
      OR      L1230  ; 進料牙插移載位置01出料側
      OUT     M1240  ; 牙插移載位置01燈
1137  LD      SM400  ; Run On
      MOV     H100 D1220  ; 定位型態
      DMOV    ZR1210 D1224  ; 牙插移載速度01 / Command  speed
      DMOV    ZR1212 D1226  ; Position address
1144  LD      L3650  ; 進料手動允許信號
      ANI     L1231  ; 牙插移載位置02  進料側
      AND     M7601  ; Run Off
      OUT     L1291  ; 允許托框回原點移載往位置02*
1148  LD      M1221  ; 牙插移載位置02 SW
      OR      L1291  ; 允許托框回原點移載往位置02*
      AND     L4509  ; 進料牙叉下定點
      AND     L1230  ; 進料牙插移載位置01出料側
      AND     L3650  ; 進料手動允許信號
      AND     B2D  ; 連線上游出板要求
      OUT     T1221 K10  ; 牙插移載位置02延遲
1158  LD      L3660  ; 進料啟動允許信號
      OR      L3670  ; 進料測試允許信號
      LD      L3794  ; 每段設定溫度到達
      OR      L200  ; 加熱不連鎖
      ANB
      AND     M5100  ; 進料手臂自動啟動SW燈
      AND     L4504  ; 進料牙叉夾板    開定點
      AND     L4507  ; 進料牙叉無板檢知
      AND     L4509  ; 進料牙叉下定點
      ANI     L1231  ; 牙插移載位置02  進料側
      AND     L1230  ; 進料牙插移載位置01出料側
      ANI     L1231  ; 牙插移載位置02  進料側
      ANI     L3601  ; 停止中  信號
      AND     B2D  ; 連線上游出板要求
      ANI     M7062  ; 上位停止放板KP
      ANI     B3342  ; 進料連線取消
      OUT     T1251 D118  ; 牙插移載位置自動往  位置02 / 伺服機構自動運轉延遲時間
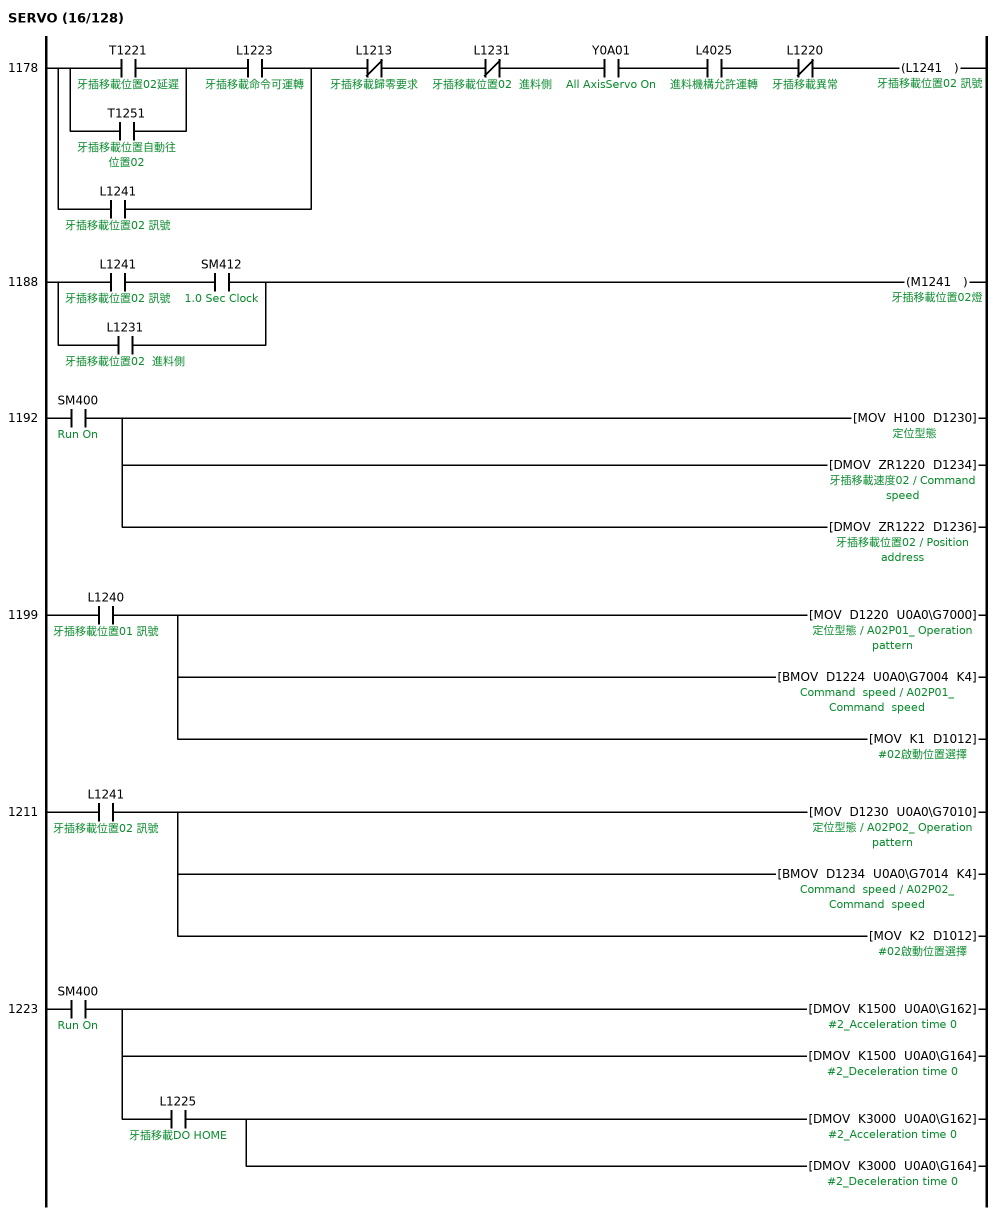
1178  LD      T1221  ; 牙插移載位置02延遲
      OR      T1251  ; 牙插移載位置自動往  位置02
      AND     L1223  ; 牙插移載命令可運轉
      OR      L1241  ; 牙插移載位置02 訊號
      ANI     L1213  ; 牙插移載歸零要求
      ANI     L1231  ; 牙插移載位置02  進料側
      AND     Y0A01  ; All AxisServo On
      AND     L4025  ; 進料機構允許運轉
      ANI     L1220  ; 牙插移載異常
      OUT     L1241  ; 牙插移載位置02 訊號
1188  LD      L1241  ; 牙插移載位置02 訊號
      AND     SM412  ; 1.0 Sec Clock
      OR      L1231  ; 牙插移載位置02  進料側
      OUT     M1241  ; 牙插移載位置02燈
1192  LD      SM400  ; Run On
      MOV     H100 D1230  ; 定位型態
      DMOV    ZR1220 D1234  ; 牙插移載速度02 / Command  speed
      DMOV    ZR1222 D1236  ; Position address
1199  LD      L1240  ; 牙插移載位置01 訊號
      MOV     D1220 U0A0\G7000  ; A02P01_ Operation pattern
      BMOV    D1224 U0A0\G7004 K4  ; A02P01_ Command  speed
      MOV     K1 D1012  ; #02啟動位置選擇
1211  LD      L1241  ; 牙插移載位置02 訊號
      MOV     D1230 U0A0\G7010  ; A02P02_ Operation pattern
      BMOV    D1234 U0A0\G7014 K4  ; A02P02_ Command  speed
      MOV     K2 D1012
1223  LD      SM400  ; Run On
      DMOV    K1500 U0A0\G162  ; #2_Acceleration time 0
      DMOV    K1500 U0A0\G164  ; #2_Deceleration time 0
      AND     L1225  ; 牙插移載DO HOME
      DMOV    K3000 U0A0\G162
      DMOV    K3000 U0A0\G164
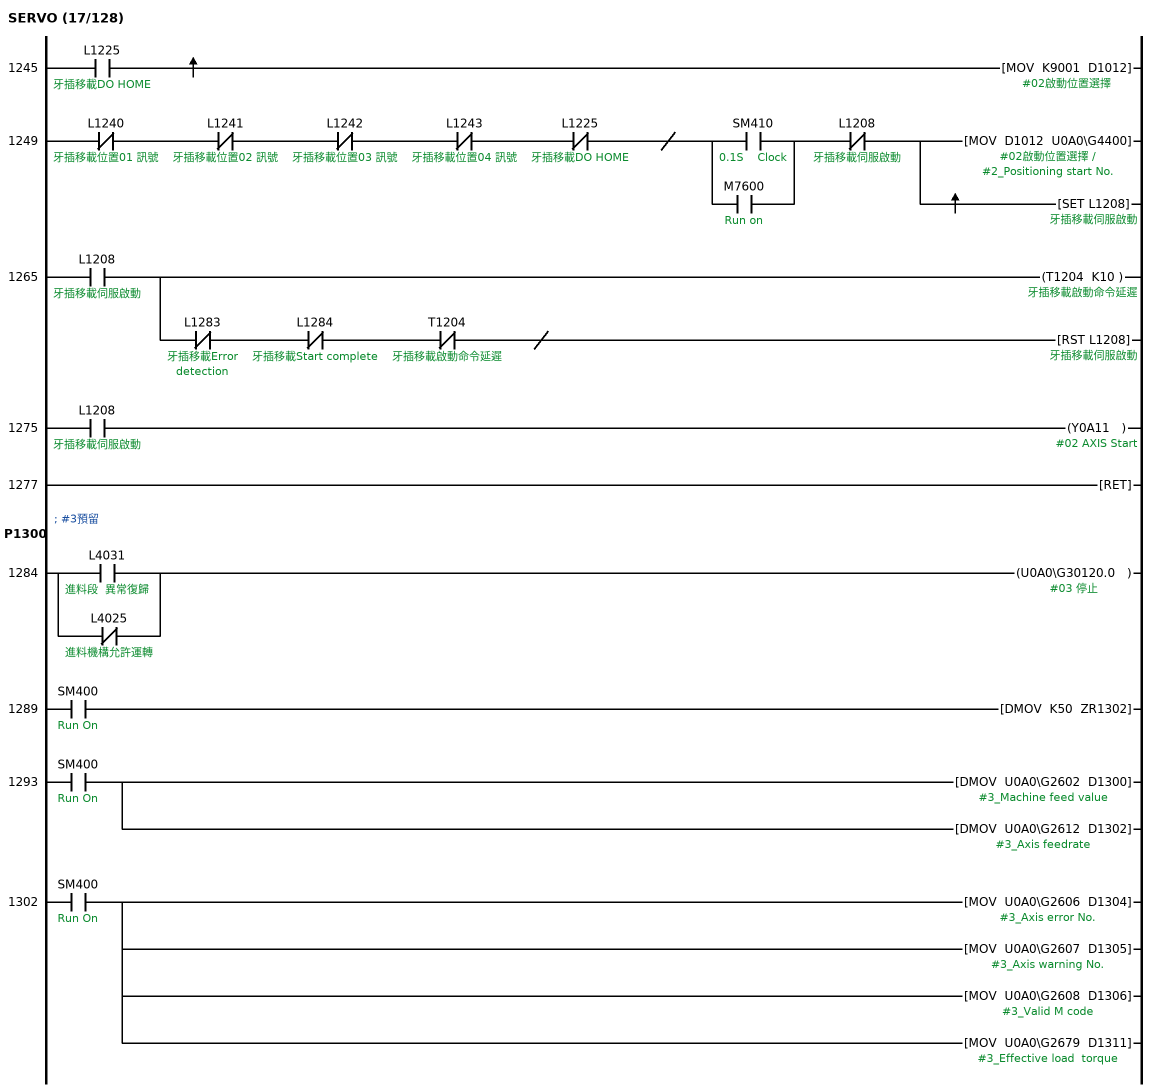
1245  LD      L1225  ; 牙插移載DO HOME
      MEP
      MOV     K9001 D1012
1249  LDI     L1240  ; 牙插移載位置01 訊號
      ANI     L1241  ; 牙插移載位置02 訊號
      ANI     L1242  ; 牙插移載位置03 訊號
      ANI     L1243  ; 牙插移載位置04 訊號
      ANI     L1225  ; 牙插移載DO HOME
      INV
      LD      SM410  ; 0.1S    Clock
      OR      M7600  ; Run on
      ANB
      ANI     L1208  ; 牙插移載伺服啟動
      MOV     D1012 U0A0\G4400  ; #2_Positioning start No.
      MEP
      SET     L1208  ; 牙插移載伺服啟動
1265  LD      L1208  ; 牙插移載伺服啟動
      OUT     T1204 K10  ; 牙插移載啟動命令延遲
      ANI     L1283  ; 牙插移載Error detection
      ANI     L1284  ; 牙插移載Start complete
      ANI     T1204  ; 牙插移載啟動命令延遲
      INV
      RST     L1208  ; 牙插移載伺服啟動
1275  LD      L1208  ; 牙插移載伺服啟動
      OUT     Y0A11  ; #02 AXIS Start
1277  RET
      P1300
; #3預留
1284  LD      L4031  ; 進料段  異常復歸
      ORI     L4025  ; 進料機構允許運轉
      OUT     U0A0\G30120.0  ; #03 停止
1289  LD      SM400  ; Run On
      DMOV    K50 ZR1302
1293  LD      SM400  ; Run On
      DMOV    U0A0\G2602 D1300  ; #3_Machine feed value
      DMOV    U0A0\G2612 D1302  ; #3_Axis feedrate
1302  LD      SM400  ; Run On
      MOV     U0A0\G2606 D1304  ; #3_Axis error No.
      MOV     U0A0\G2607 D1305  ; #3_Axis warning No.
      MOV     U0A0\G2608 D1306  ; #3_Valid M code
      MOV     U0A0\G2679 D1311  ; #3_Effective load  torque
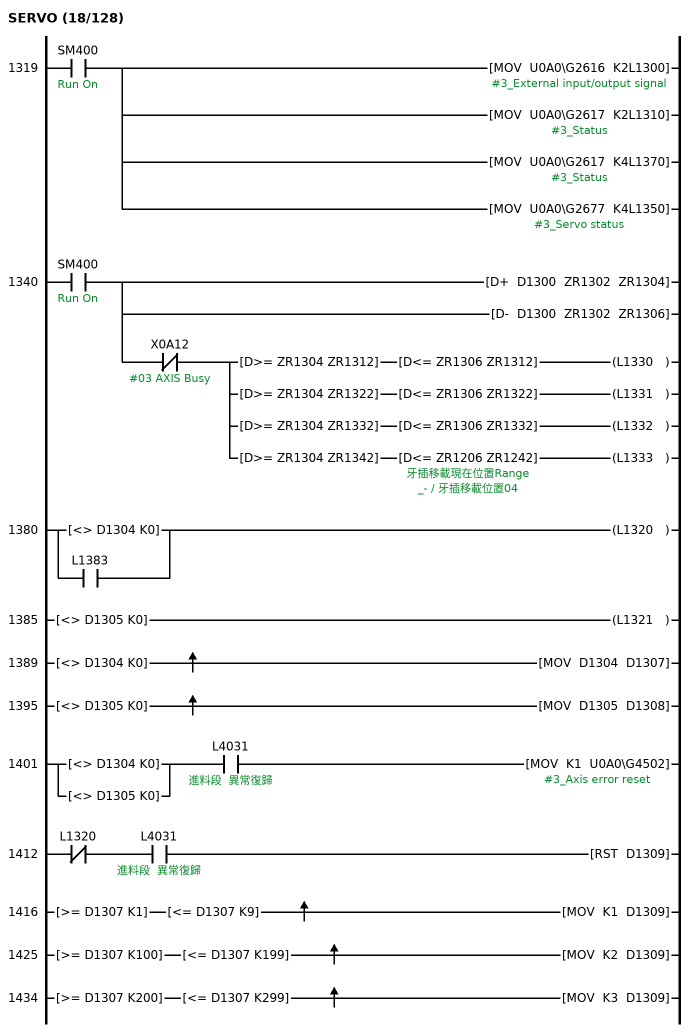
1319  LD      SM400  ; Run On
      MOV     U0A0\G2616 K2L1300  ; #3_External input/output signal
      MOV     U0A0\G2617 K2L1310  ; #3_Status
      MOV     U0A0\G2617 K4L1370
      MOV     U0A0\G2677 K4L1350  ; #3_Servo status
1340  LD      SM400  ; Run On
      D+      D1300 ZR1302 ZR1304
      D-      D1300 ZR1302 ZR1306
      ANI     X0A12  ; #03 AXIS Busy
      MPS
      ANDD>=  ZR1304 ZR1312
      ANDD<=  ZR1306 ZR1312
      OUT     L1330
      MRD
      ANDD>=  ZR1304 ZR1322
      ANDD<=  ZR1306 ZR1322
      OUT     L1331
      MRD
      ANDD>=  ZR1304 ZR1332
      ANDD<=  ZR1306 ZR1332
      OUT     L1332
      MPP
      ANDD>=  ZR1304 ZR1342
      ANDD<=  ZR1206 ZR1242  ; 牙插移載現在位置Range_- / 牙插移載位置04
      OUT     L1333
1380  LD<>    D1304 K0
      OR      L1383
      OUT     L1320
1385  LD<>    D1305 K0
      OUT     L1321
1389  LD<>    D1304 K0
      MEP
      MOV     D1304 D1307
1395  LD<>    D1305 K0
      MEP
      MOV     D1305 D1308
1401  LD<>    D1304 K0
      OR<>    D1305 K0
      AND     L4031  ; 進料段  異常復歸
      MOV     K1 U0A0\G4502  ; #3_Axis error reset
1412  LDI     L1320
      AND     L4031  ; 進料段  異常復歸
      RST     D1309
1416  LD>=    D1307 K1
      AND<=   D1307 K9
      MEP
      MOV     K1 D1309
1425  LD>=    D1307 K100
      AND<=   D1307 K199
      MEP
      MOV     K2 D1309
1434  LD>=    D1307 K200
      AND<=   D1307 K299
      MEP
      MOV     K3 D1309
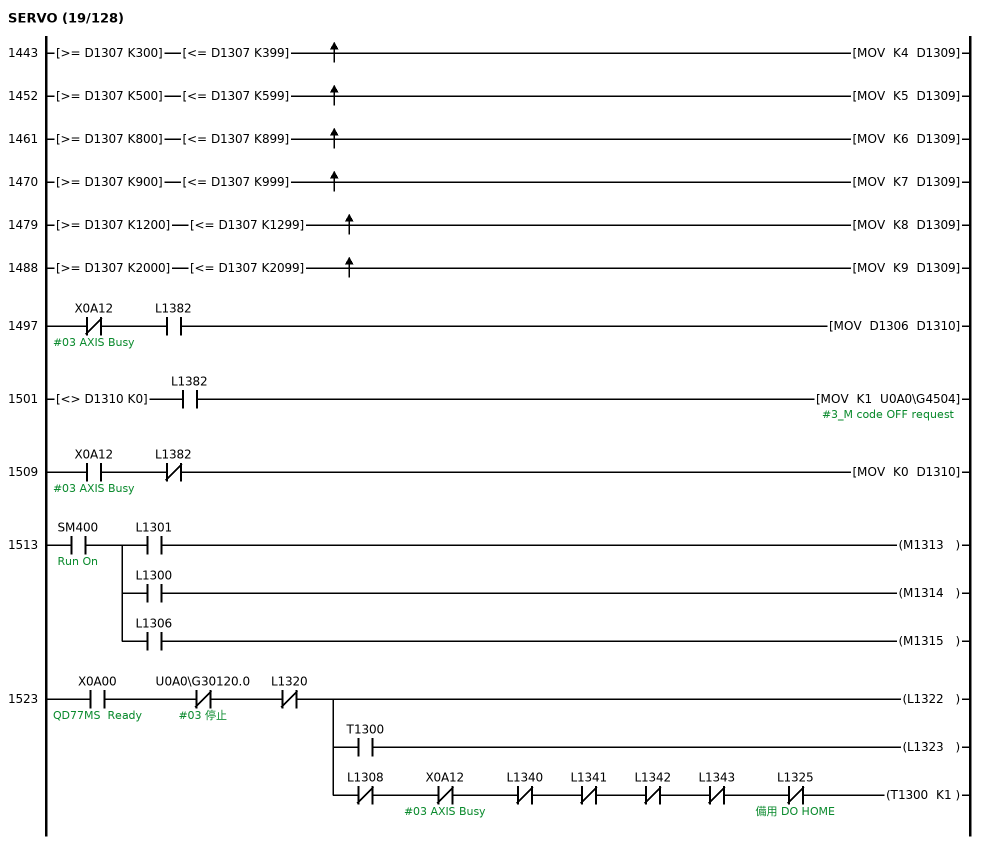
1443  LD>=    D1307 K300
      AND<=   D1307 K399
      MEP
      MOV     K4 D1309
1452  LD>=    D1307 K500
      AND<=   D1307 K599
      MEP
      MOV     K5 D1309
1461  LD>=    D1307 K800
      AND<=   D1307 K899
      MEP
      MOV     K6 D1309
1470  LD>=    D1307 K900
      AND<=   D1307 K999
      MEP
      MOV     K7 D1309
1479  LD>=    D1307 K1200
      AND<=   D1307 K1299
      MEP
      MOV     K8 D1309
1488  LD>=    D1307 K2000
      AND<=   D1307 K2099
      MEP
      MOV     K9 D1309
1497  LDI     X0A12  ; #03 AXIS Busy
      AND     L1382
      MOV     D1306 D1310
1501  LD<>    D1310 K0
      AND     L1382
      MOV     K1 U0A0\G4504  ; #3_M code OFF request
1509  LD      X0A12  ; #03 AXIS Busy
      ANI     L1382
      MOV     K0 D1310
1513  LD      SM400  ; Run On
      MPS
      AND     L1301
      OUT     M1313
      MRD
      AND     L1300
      OUT     M1314
      MPP
      AND     L1306
      OUT     M1315
1523  LD      X0A00  ; QD77MS  Ready
      ANI     U0A0\G30120.0  ; #03 停止
      ANI     L1320
      OUT     L1322
      MPS
      AND     T1300
      OUT     L1323
      MPP
      ANI     L1308
      ANI     X0A12  ; #03 AXIS Busy
      ANI     L1340
      ANI     L1341
      ANI     L1342
      ANI     L1343
      ANI     L1325  ; 備用 DO HOME
      OUT     T1300 K1
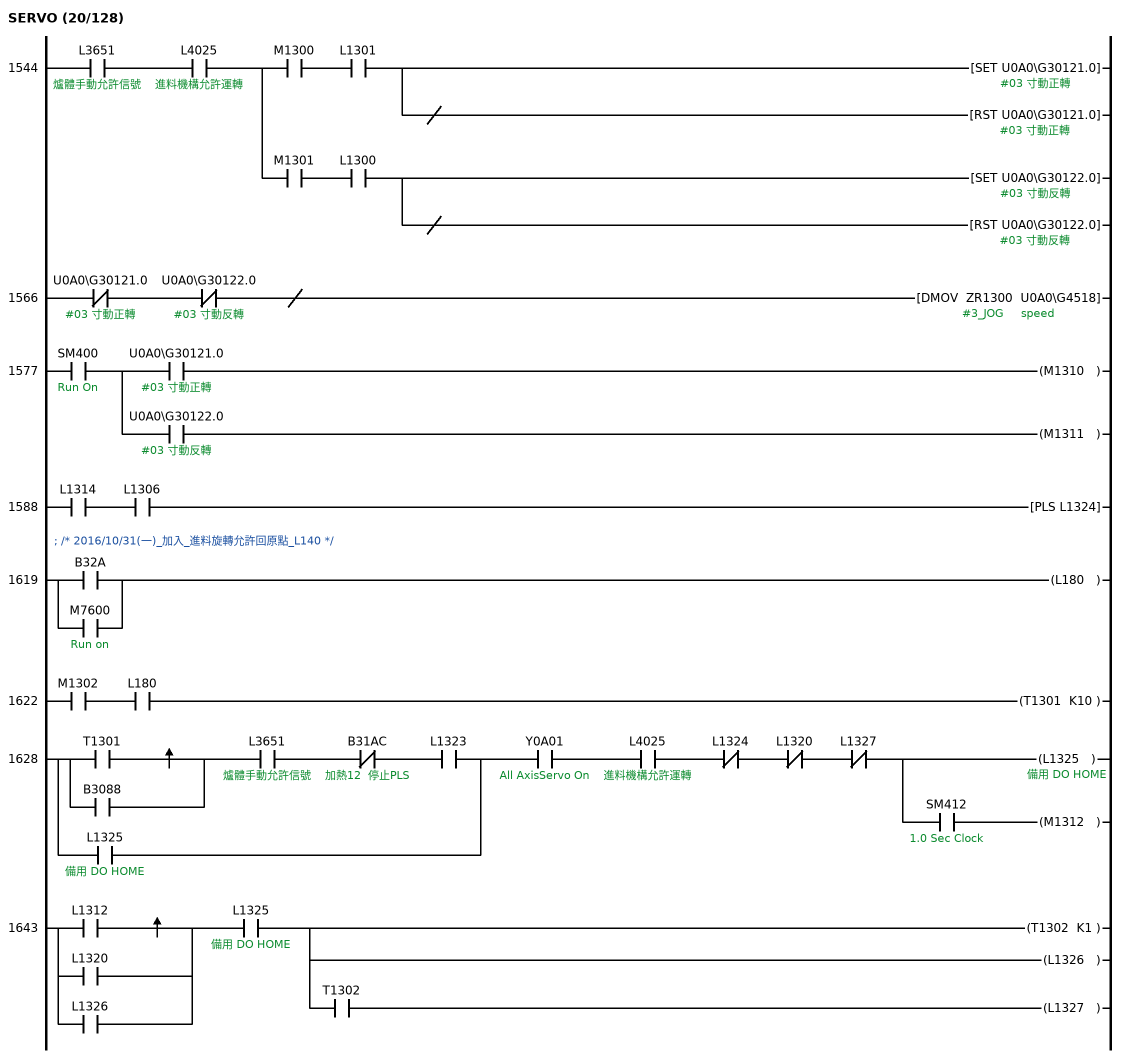
1544  LD      L3651  ; 爐體手動允許信號
      AND     L4025  ; 進料機構允許運轉
      MPS
      AND     M1300
      AND     L1301
      SET     U0A0\G30121.0  ; #03 寸動正轉
      INV
      RST     U0A0\G30121.0  ; #03 寸動正轉
      MPP
      AND     M1301
      AND     L1300
      SET     U0A0\G30122.0  ; #03 寸動反轉
      INV
      RST     U0A0\G30122.0  ; #03 寸動反轉
1566  LDI     U0A0\G30121.0  ; #03 寸動正轉
      ANI     U0A0\G30122.0  ; #03 寸動反轉
      INV
      DMOV    ZR1300 U0A0\G4518  ; #3_JOG     speed
1577  LD      SM400  ; Run On
      MPS
      AND     U0A0\G30121.0  ; #03 寸動正轉
      OUT     M1310
      MPP
      AND     U0A0\G30122.0  ; #03 寸動反轉
      OUT     M1311
1588  LD      L1314
      AND     L1306
      PLS     L1324
; /* 2016/10/31(一)_加入_進料旋轉允許回原點_L140 */
1619  LD      B32A
      OR      M7600  ; Run on
      OUT     L180
1622  LD      M1302
      AND     L180
      OUT     T1301 K10
1628  LD      T1301
      MEP
      OR      B3088
      AND     L3651  ; 爐體手動允許信號
      ANI     B31AC  ; 加熱12  停止PLS
      AND     L1323
      OR      L1325  ; 備用 DO HOME
      AND     Y0A01  ; All AxisServo On
      AND     L4025  ; 進料機構允許運轉
      ANI     L1324
      ANI     L1320
      ANI     L1327
      OUT     L1325  ; 備用 DO HOME
      AND     SM412  ; 1.0 Sec Clock
      OUT     M1312
1643  LD      L1312
      MEP
      OR      L1320
      OR      L1326
      AND     L1325  ; 備用 DO HOME
      OUT     T1302 K1
      OUT     L1326
      AND     T1302
      OUT     L1327
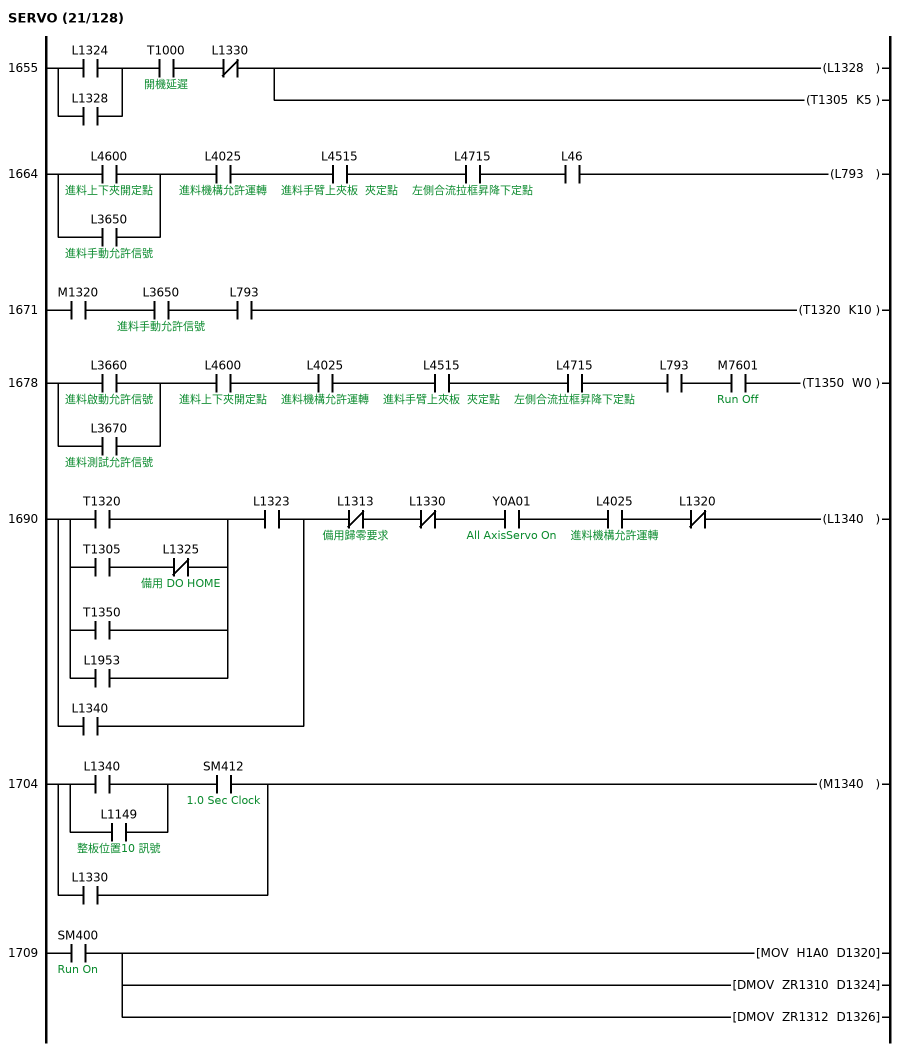
1655  LD      L1324
      OR      L1328
      AND     T1000  ; 開機延遲
      ANI     L1330
      OUT     L1328
      OUT     T1305 K5
1664  LD      L4600  ; 進料上下夾開定點
      OR      L3650  ; 進料手動允許信號
      AND     L4025  ; 進料機構允許運轉
      AND     L4515  ; 進料手臂上夾板  夾定點
      AND     L4715  ; 左側合流拉框昇降下定點
      AND     L46
      OUT     L793
1671  LD      M1320
      AND     L3650  ; 進料手動允許信號
      AND     L793
      OUT     T1320 K10
1678  LD      L3660  ; 進料啟動允許信號
      OR      L3670  ; 進料測試允許信號
      AND     L4600  ; 進料上下夾開定點
      AND     L4025  ; 進料機構允許運轉
      AND     L4515  ; 進料手臂上夾板  夾定點
      AND     L4715  ; 左側合流拉框昇降下定點
      AND     L793
      AND     M7601  ; Run Off
      OUT     T1350 W0
1690  LD      T1320
      LD      T1305
      ANI     L1325  ; 備用 DO HOME
      ORB
      OR      T1350
      OR      L1953
      AND     L1323
      OR      L1340
      ANI     L1313  ; 備用歸零要求
      ANI     L1330
      AND     Y0A01  ; All AxisServo On
      AND     L4025  ; 進料機構允許運轉
      ANI     L1320
      OUT     L1340
1704  LD      L1340
      OR      L1149  ; 整板位置10 訊號
      AND     SM412  ; 1.0 Sec Clock
      OR      L1330
      OUT     M1340
1709  LD      SM400  ; Run On
      MOV     H1A0 D1320
      DMOV    ZR1310 D1324
      DMOV    ZR1312 D1326
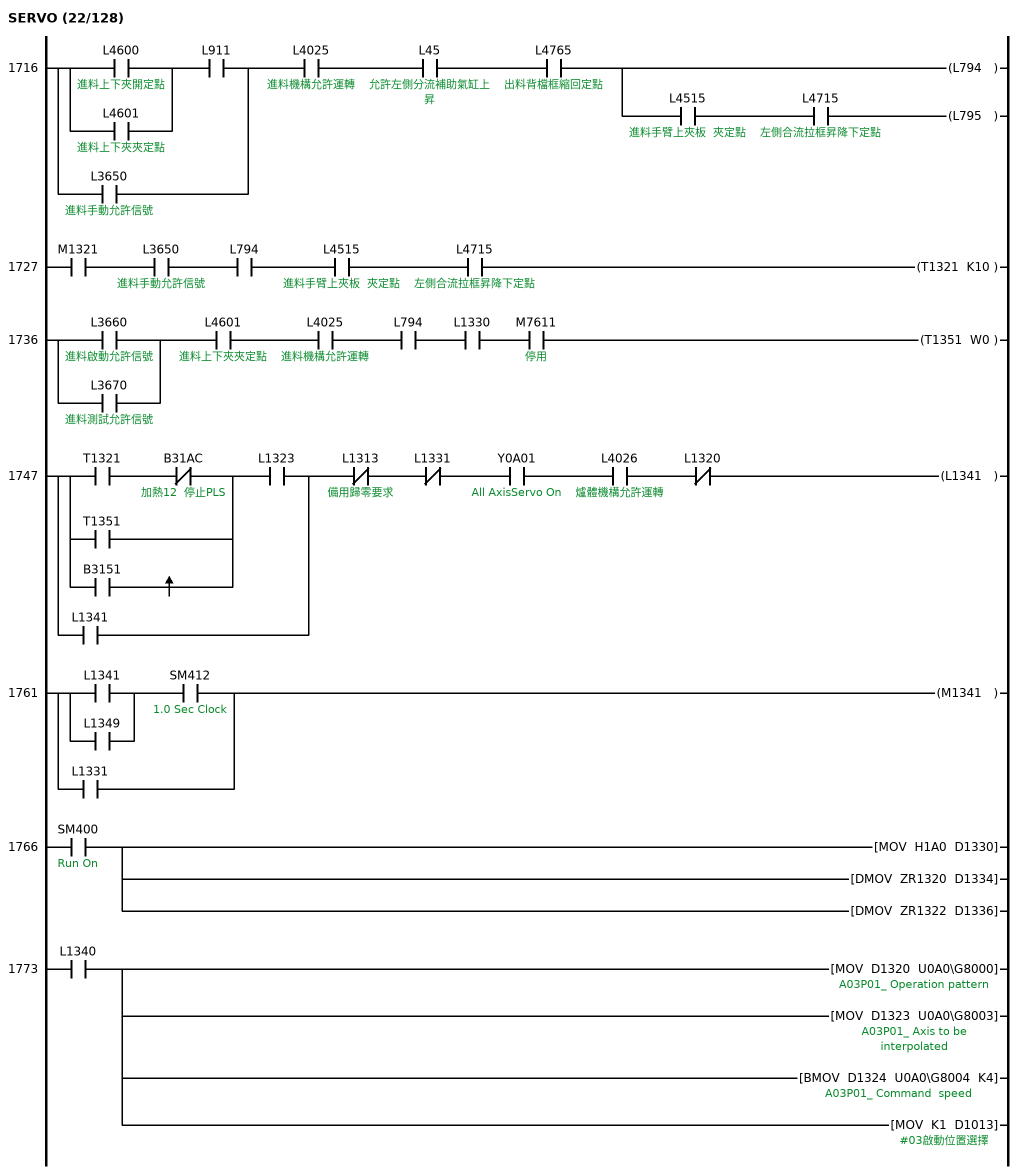
1716  LD      L4600  ; 進料上下夾開定點
      OR      L4601  ; 進料上下夾夾定點
      AND     L911
      OR      L3650  ; 進料手動允許信號
      AND     L4025  ; 進料機構允許運轉
      AND     L45  ; 允許左側分流補助氣缸上昇
      AND     L4765  ; 出料背檔框縮回定點
      OUT     L794
      AND     L4515  ; 進料手臂上夾板  夾定點
      AND     L4715  ; 左側合流拉框昇降下定點
      OUT     L795
1727  LD      M1321
      AND     L3650  ; 進料手動允許信號
      AND     L794
      AND     L4515  ; 進料手臂上夾板  夾定點
      AND     L4715  ; 左側合流拉框昇降下定點
      OUT     T1321 K10
1736  LD      L3660  ; 進料啟動允許信號
      OR      L3670  ; 進料測試允許信號
      AND     L4601  ; 進料上下夾夾定點
      AND     L4025  ; 進料機構允許運轉
      AND     L794
      AND     L1330
      AND     M7611  ; 停用
      OUT     T1351 W0
1747  LD      T1321
      ANI     B31AC  ; 加熱12  停止PLS
      OR      T1351
      LD      B3151
      MEP
      ORB
      AND     L1323
      OR      L1341
      ANI     L1313  ; 備用歸零要求
      ANI     L1331
      AND     Y0A01  ; All AxisServo On
      AND     L4026  ; 爐體機構允許運轉
      ANI     L1320
      OUT     L1341
1761  LD      L1341
      OR      L1349
      AND     SM412  ; 1.0 Sec Clock
      OR      L1331
      OUT     M1341
1766  LD      SM400  ; Run On
      MOV     H1A0 D1330
      DMOV    ZR1320 D1334
      DMOV    ZR1322 D1336
1773  LD      L1340
      MOV     D1320 U0A0\G8000  ; A03P01_ Operation pattern
      MOV     D1323 U0A0\G8003  ; A03P01_ Axis to be interpolated
      BMOV    D1324 U0A0\G8004 K4  ; A03P01_ Command  speed
      MOV     K1 D1013  ; #03啟動位置選擇
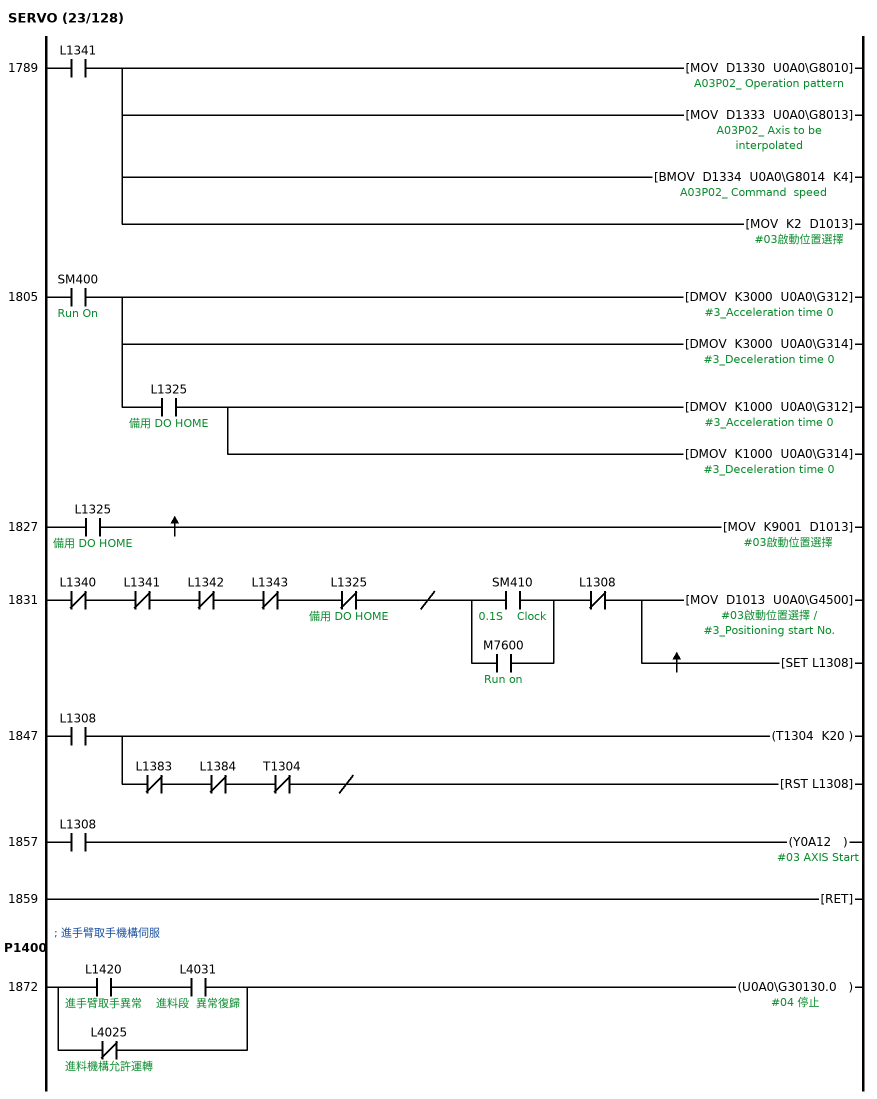
1789  LD      L1341
      MOV     D1330 U0A0\G8010  ; A03P02_ Operation pattern
      MOV     D1333 U0A0\G8013  ; A03P02_ Axis to be interpolated
      BMOV    D1334 U0A0\G8014 K4  ; A03P02_ Command  speed
      MOV     K2 D1013
1805  LD      SM400  ; Run On
      DMOV    K3000 U0A0\G312  ; #3_Acceleration time 0
      DMOV    K3000 U0A0\G314  ; #3_Deceleration time 0
      AND     L1325  ; 備用 DO HOME
      DMOV    K1000 U0A0\G312
      DMOV    K1000 U0A0\G314
1827  LD      L1325  ; 備用 DO HOME
      MEP
      MOV     K9001 D1013
1831  LDI     L1340
      ANI     L1341
      ANI     L1342
      ANI     L1343
      ANI     L1325  ; 備用 DO HOME
      INV
      LD      SM410  ; 0.1S    Clock
      OR      M7600  ; Run on
      ANB
      ANI     L1308
      MOV     D1013 U0A0\G4500  ; #3_Positioning start No.
      MEP
      SET     L1308
1847  LD      L1308
      OUT     T1304 K20
      ANI     L1383
      ANI     L1384
      ANI     T1304
      INV
      RST     L1308
1857  LD      L1308
      OUT     Y0A12  ; #03 AXIS Start
1859  RET
      P1400
; 進手臂取手機構伺服
1872  LD      L1420  ; 進手臂取手異常
      AND     L4031  ; 進料段  異常復歸
      ORI     L4025  ; 進料機構允許運轉
      OUT     U0A0\G30130.0  ; #04 停止
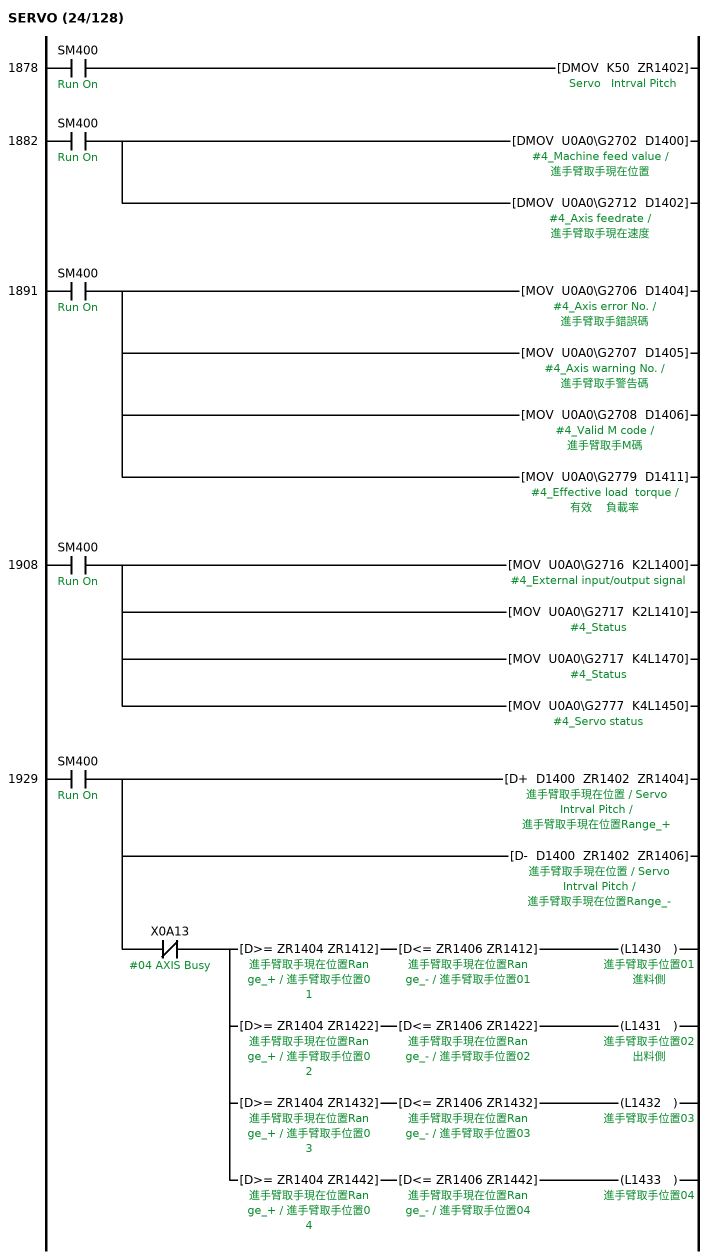
1878  LD      SM400  ; Run On
      DMOV    K50 ZR1402  ; Servo   Intrval Pitch
1882  LD      SM400  ; Run On
      DMOV    U0A0\G2702 D1400  ; #4_Machine feed value / 進手臂取手現在位置
      DMOV    U0A0\G2712 D1402  ; #4_Axis feedrate / 進手臂取手現在速度
1891  LD      SM400  ; Run On
      MOV     U0A0\G2706 D1404  ; #4_Axis error No. / 進手臂取手錯誤碼
      MOV     U0A0\G2707 D1405  ; #4_Axis warning No. / 進手臂取手警告碼
      MOV     U0A0\G2708 D1406  ; #4_Valid M code / 進手臂取手M碼
      MOV     U0A0\G2779 D1411  ; #4_Effective load  torque / 有效    負載率
1908  LD      SM400  ; Run On
      MOV     U0A0\G2716 K2L1400  ; #4_External input/output signal / 進手臂取手    負極限
      MOV     U0A0\G2717 K2L1410  ; #4_Status / 進手臂取手速度控制
      MOV     U0A0\G2717 K4L1470  ; 進手臂取手速度控制
      MOV     U0A0\G2777 K4L1450  ; #4_Servo status / READY ON
1929  LD      SM400  ; Run On
      D+      D1400 ZR1402 ZR1404  ; 進手臂取手現在位置Range_+
      D-      D1400 ZR1402 ZR1406  ; 進手臂取手現在位置Range_-
      ANI     X0A13  ; #04 AXIS Busy
      MPS
      ANDD>=  ZR1404 ZR1412  ; 進手臂取手現在位置Range_+ / 進手臂取手位置01
      ANDD<=  ZR1406 ZR1412  ; 進手臂取手現在位置Range_- / 進手臂取手位置01
      OUT     L1430  ; 進手臂取手位置01  進料側
      MRD
      ANDD>=  ZR1404 ZR1422  ; 進手臂取手現在位置Range_+ / 進手臂取手位置02
      ANDD<=  ZR1406 ZR1422  ; 進手臂取手現在位置Range_- / 進手臂取手位置02
      OUT     L1431  ; 進手臂取手位置02  出料側
      MRD
      ANDD>=  ZR1404 ZR1432  ; 進手臂取手現在位置Range_+ / 進手臂取手位置03
      ANDD<=  ZR1406 ZR1432  ; 進手臂取手現在位置Range_- / 進手臂取手位置03
      OUT     L1432  ; 進手臂取手位置03
      MPP
      ANDD>=  ZR1404 ZR1442  ; 進手臂取手現在位置Range_+ / 進手臂取手位置04
      ANDD<=  ZR1406 ZR1442  ; 進手臂取手現在位置Range_- / 進手臂取手位置04
      OUT     L1433  ; 進手臂取手位置04
